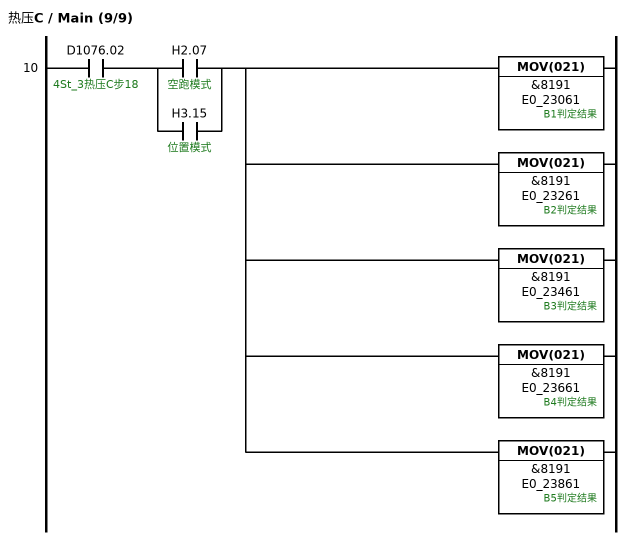
; [picture p216: 热压C / Main, rungs 10-10]
; rung 10
LD D1076.02  ; 4St_3热压C步18
LD H2.07  ; 空跑模式
OR H3.15  ; 位置模式
ANDLD
MOV(021) &8191 E0_23061  ; B1判定结果
MOV(021) &8191 E0_23261  ; B2判定结果
MOV(021) &8191 E0_23461  ; B3判定结果
MOV(021) &8191 E0_23661  ; B4判定结果
MOV(021) &8191 E0_23861  ; B5判定结果

### Section _4ST_3热压C

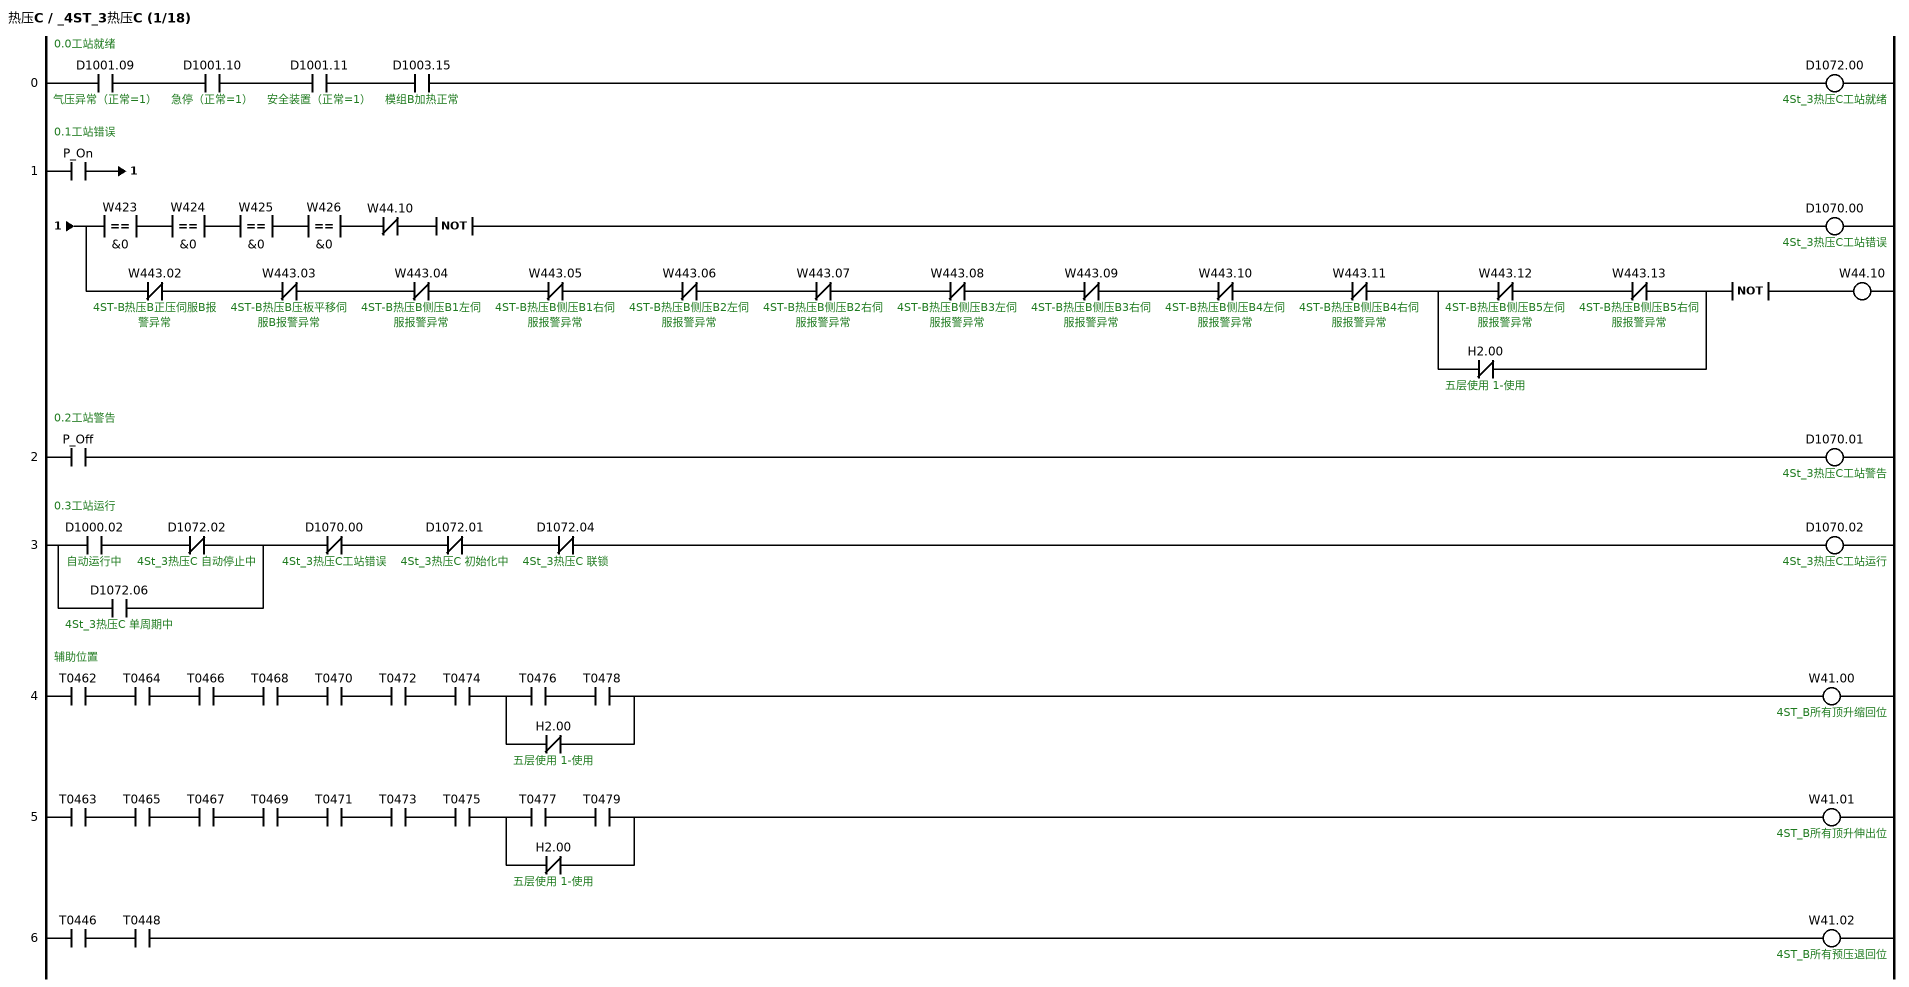
; rung 0: 0.0工站就绪
LD D1001.09  ; 气压异常（正常=1）
AND D1001.10  ; 急停（正常=1）
AND D1001.11  ; 安全装置（正常=1）
AND D1003.15  ; 模组B加热正常
OUT D1072.00  ; 4St_3热压C工站就绪
; rung 1: 0.1工站错误
LD P_On
OUT TR0
AND=(300) W423 &0
AND=(300) W424 &0
AND=(300) W425 &0
AND=(300) W426 &0
ANDNOT W44.10
NOT(520)
OUT D1070.00  ; 4St_3热压C工站错误
LD TR0
ANDNOT W443.02  ; 4ST-B热压B正压伺服B报警异常
ANDNOT W443.03  ; 4ST-B热压B压板平移伺服B报警异常
ANDNOT W443.04  ; 4ST-B热压B侧压B1左伺服报警异常
ANDNOT W443.05  ; 4ST-B热压B侧压B1右伺服报警异常
ANDNOT W443.06  ; 4ST-B热压B侧压B2左伺服报警异常
ANDNOT W443.07  ; 4ST-B热压B侧压B2右伺服报警异常
ANDNOT W443.08  ; 4ST-B热压B侧压B3左伺服报警异常
ANDNOT W443.09  ; 4ST-B热压B侧压B3右伺服报警异常
ANDNOT W443.10  ; 4ST-B热压B侧压B4左伺服报警异常
ANDNOT W443.11  ; 4ST-B热压B侧压B4右伺服报警异常
LDNOT W443.12  ; 4ST-B热压B侧压B5左伺服报警异常
ANDNOT W443.13  ; 4ST-B热压B侧压B5右伺服报警异常
ORNOT H2.00  ; 五层使用 1-使用
ANDLD
NOT(520)
OUT W44.10
; rung 2: 0.2工站警告
LD P_Off
OUT D1070.01  ; 4St_3热压C工站警告
; rung 3: 0.3工站运行
LD D1000.02  ; 自动运行中
ANDNOT D1072.02  ; 4St_3热压C 自动停止中
OR D1072.06  ; 4St_3热压C 单周期中
ANDNOT D1070.00  ; 4St_3热压C工站错误
ANDNOT D1072.01  ; 4St_3热压C 初始化中
ANDNOT D1072.04  ; 4St_3热压C 联锁
OUT D1070.02  ; 4St_3热压C工站运行
; rung 4: 辅助位置
LD T0462
AND T0464
AND T0466
AND T0468
AND T0470
AND T0472
AND T0474
LD T0476
AND T0478
ORNOT H2.00  ; 五层使用 1-使用
ANDLD
OUT W41.00  ; 4ST_B所有顶升缩回位
; rung 5
LD T0463
AND T0465
AND T0467
AND T0469
AND T0471
AND T0473
AND T0475
LD T0477
AND T0479
ORNOT H2.00  ; 五层使用 1-使用
ANDLD
OUT W41.01  ; 4ST_B所有顶升伸出位
; rung 6
LD T0446
AND T0448
OUT W41.02  ; 4ST_B所有预压退回位

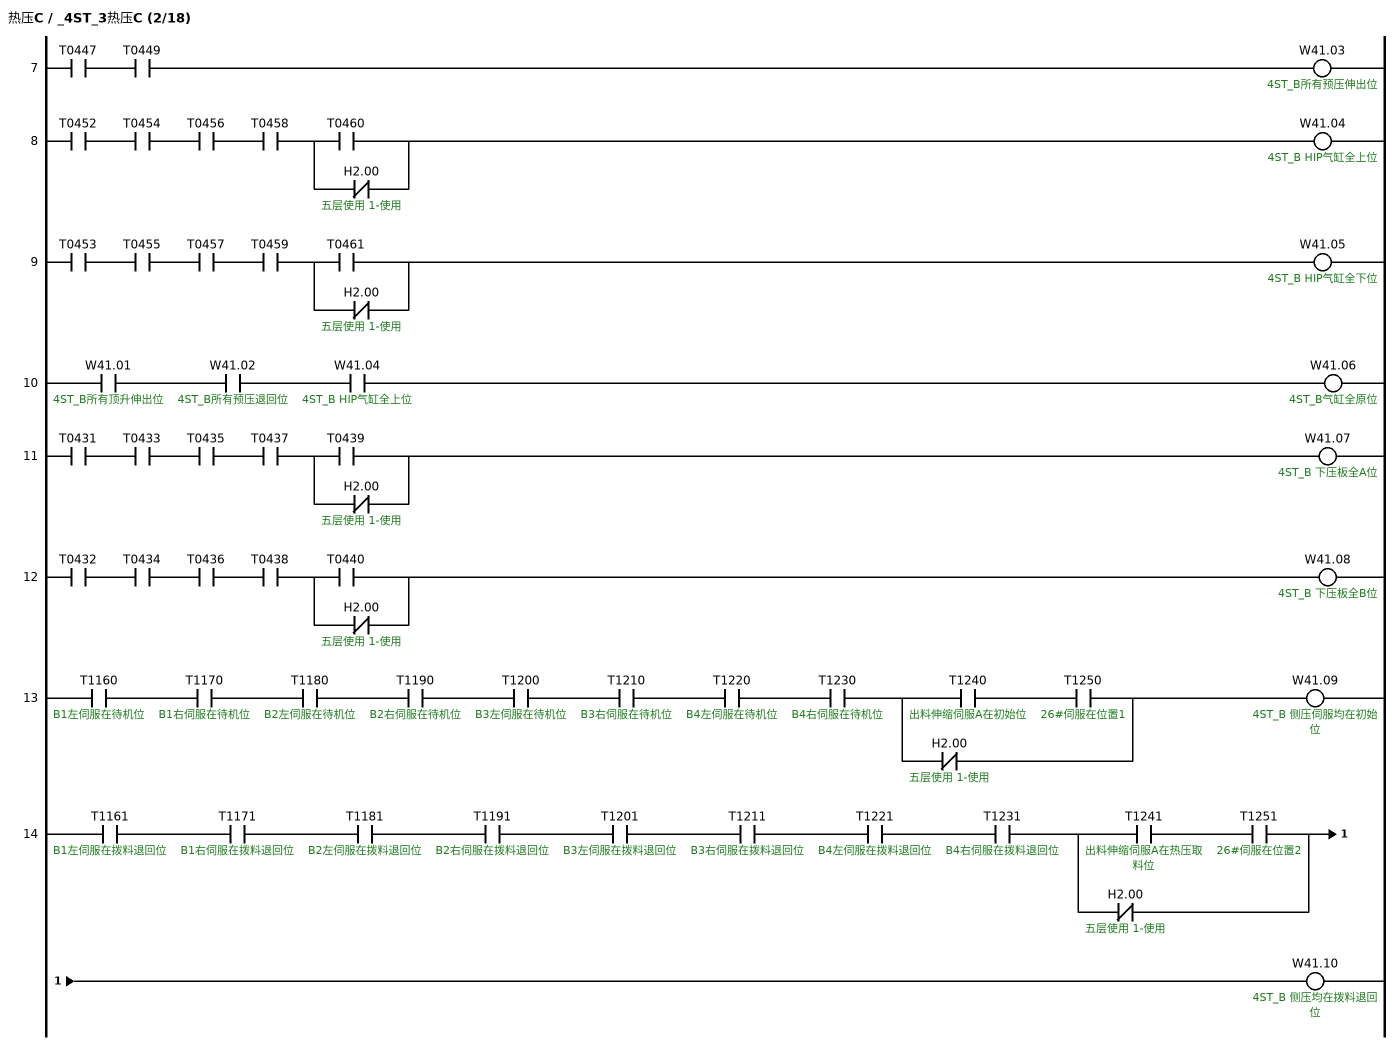
; rung 7
LD T0447
AND T0449
OUT W41.03  ; 4ST_B所有预压伸出位
; rung 8
LD T0452
AND T0454
AND T0456
AND T0458
LD T0460
ORNOT H2.00  ; 五层使用 1-使用
ANDLD
OUT W41.04  ; 4ST_B HIP气缸全上位
; rung 9
LD T0453
AND T0455
AND T0457
AND T0459
LD T0461
ORNOT H2.00  ; 五层使用 1-使用
ANDLD
OUT W41.05  ; 4ST_B HIP气缸全下位
; rung 10
LD W41.01  ; 4ST_B所有顶升伸出位
AND W41.02  ; 4ST_B所有预压退回位
AND W41.04  ; 4ST_B HIP气缸全上位
OUT W41.06  ; 4ST_B气缸全原位
; rung 11
LD T0431
AND T0433
AND T0435
AND T0437
LD T0439
ORNOT H2.00  ; 五层使用 1-使用
ANDLD
OUT W41.07  ; 4ST_B 下压板全A位
; rung 12
LD T0432
AND T0434
AND T0436
AND T0438
LD T0440
ORNOT H2.00  ; 五层使用 1-使用
ANDLD
OUT W41.08  ; 4ST_B 下压板全B位
; rung 13
LD T1160  ; B1左伺服在待机位
AND T1170  ; B1右伺服在待机位
AND T1180  ; B2左伺服在待机位
AND T1190  ; B2右伺服在待机位
AND T1200  ; B3左伺服在待机位
AND T1210  ; B3右伺服在待机位
AND T1220  ; B4左伺服在待机位
AND T1230  ; B4右伺服在待机位
LD T1240  ; 出料伸缩伺服A在初始位
AND T1250  ; 26#伺服在位置1
ORNOT H2.00  ; 五层使用 1-使用
ANDLD
OUT W41.09  ; 4ST_B 侧压伺服均在初始位
; rung 14
LD T1161  ; B1左伺服在拨料退回位
AND T1171  ; B1右伺服在拨料退回位
AND T1181  ; B2左伺服在拨料退回位
AND T1191  ; B2右伺服在拨料退回位
AND T1201  ; B3左伺服在拨料退回位
AND T1211  ; B3右伺服在拨料退回位
AND T1221  ; B4左伺服在拨料退回位
AND T1231  ; B4右伺服在拨料退回位
LD T1241  ; 出料伸缩伺服A在热压取料位
AND T1251  ; 26#伺服在位置2
ORNOT H2.00  ; 五层使用 1-使用
ANDLD
OUT W41.10  ; 4ST_B 侧压均在拨料退回位

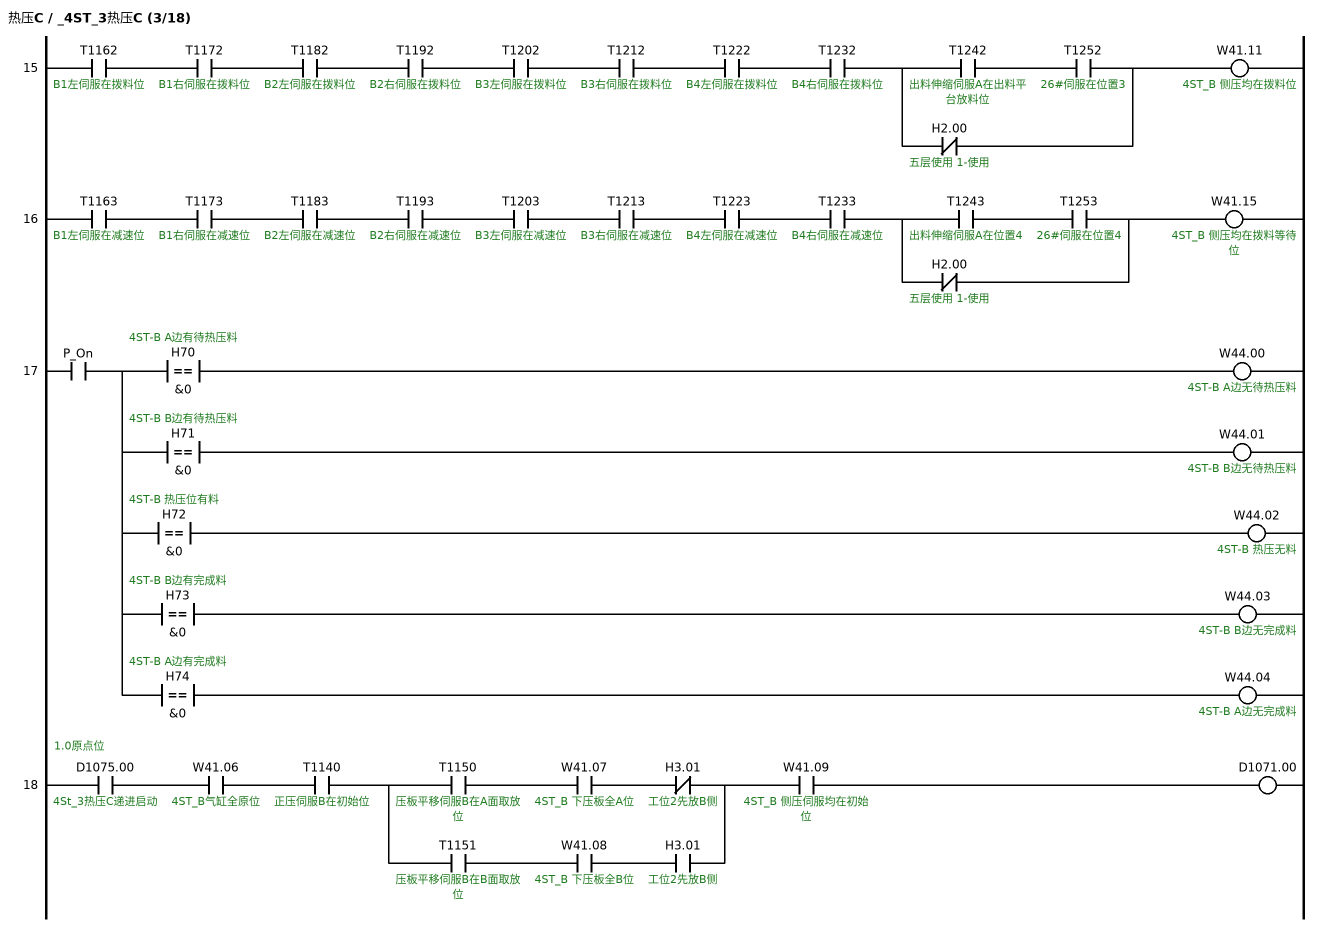
; rung 15
LD T1162  ; B1左伺服在拨料位
AND T1172  ; B1右伺服在拨料位
AND T1182  ; B2左伺服在拨料位
AND T1192  ; B2右伺服在拨料位
AND T1202  ; B3左伺服在拨料位
AND T1212  ; B3右伺服在拨料位
AND T1222  ; B4左伺服在拨料位
AND T1232  ; B4右伺服在拨料位
LD T1242  ; 出料伸缩伺服A在出料平台放料位
AND T1252  ; 26#伺服在位置3
ORNOT H2.00  ; 五层使用 1-使用
ANDLD
OUT W41.11  ; 4ST_B 侧压均在拨料位
; rung 16
LD T1163  ; B1左伺服在减速位
AND T1173  ; B1右伺服在减速位
AND T1183  ; B2左伺服在减速位
AND T1193  ; B2右伺服在减速位
AND T1203  ; B3左伺服在减速位
AND T1213  ; B3右伺服在减速位
AND T1223  ; B4左伺服在减速位
AND T1233  ; B4右伺服在减速位
LD T1243  ; 出料伸缩伺服A在位置4
AND T1253  ; 26#伺服在位置4
ORNOT H2.00  ; 五层使用 1-使用
ANDLD
OUT W41.15  ; 4ST_B 侧压均在拨料等待位
; rung 17
LD P_On
OUT TR0
AND=(300) H70 &0  ; 4ST-B A边有待热压料
OUT W44.00  ; 4ST-B A边无待热压料
LD TR0
AND=(300) H71 &0  ; 4ST-B B边有待热压料
OUT W44.01  ; 4ST-B B边无待热压料
LD TR0
AND=(300) H72 &0  ; 4ST-B 热压位有料
OUT W44.02  ; 4ST-B 热压无料
LD TR0
AND=(300) H73 &0  ; 4ST-B B边有完成料
OUT W44.03  ; 4ST-B B边无完成料
LD TR0
AND=(300) H74 &0  ; 4ST-B A边有完成料
OUT W44.04  ; 4ST-B A边无完成料
; rung 18: 1.0原点位
LD D1075.00  ; 4St_3热压C递进启动
AND W41.06  ; 4ST_B气缸全原位
AND T1140  ; 正压伺服B在初始位
LD T1150  ; 压板平移伺服B在A面取放位
AND W41.07  ; 4ST_B 下压板全A位
ANDNOT H3.01  ; 工位2先放B侧
LD T1151  ; 压板平移伺服B在B面取放位
AND W41.08  ; 4ST_B 下压板全B位
AND H3.01  ; 工位2先放B侧
ORLD
ANDLD
AND W41.09  ; 4ST_B 侧压伺服均在初始位
OUT D1071.00

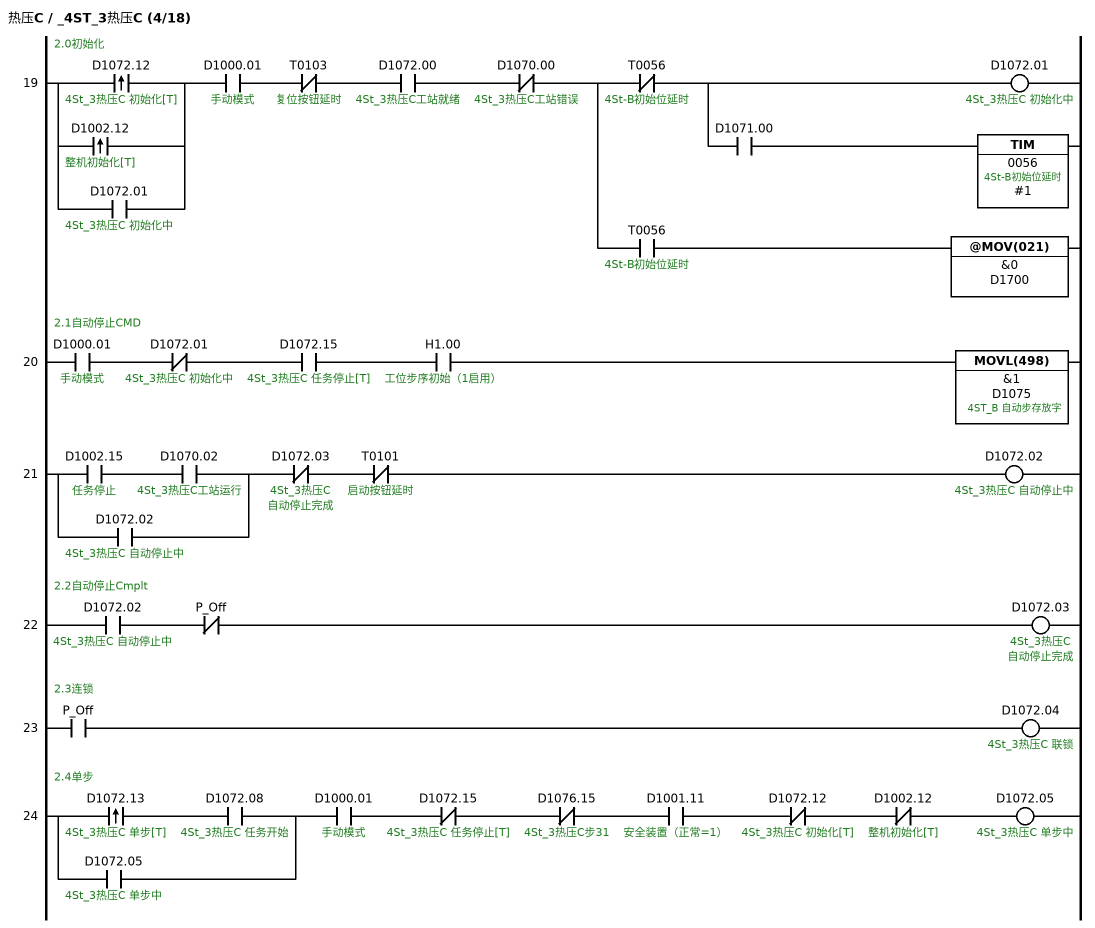
; rung 19: 2.0初始化
@LD D1072.12  ; 4St_3热压C 初始化[T]
@OR D1002.12  ; 整机初始化[T]
OR D1072.01  ; 4St_3热压C 初始化中
AND D1000.01  ; 手动模式
ANDNOT T0103  ; 复位按钮延时
AND D1072.00  ; 4St_3热压C工站就绪
ANDNOT D1070.00  ; 4St_3热压C工站错误
OUT TR0
ANDNOT T0056  ; 4St-B初始位延时
OUT D1072.01  ; 4St_3热压C 初始化中
AND D1071.00
TIM 0056 #1  ; 4St-B初始位延时
LD TR0
AND T0056  ; 4St-B初始位延时
@MOV(021) &0 D1700
; rung 20: 2.1自动停止CMD
LD D1000.01  ; 手动模式
ANDNOT D1072.01  ; 4St_3热压C 初始化中
AND D1072.15  ; 4St_3热压C 任务停止[T]
AND H1.00  ; 工位步序初始（1启用）
MOVL(498) &1 D1075  ; 4ST_B 自动步存放字
; rung 21
LD D1002.15  ; 任务停止
AND D1070.02  ; 4St_3热压C工站运行
OR D1072.02  ; 4St_3热压C 自动停止中
ANDNOT D1072.03  ; 4St_3热压C 自动停止完成
ANDNOT T0101  ; 启动按钮延时
OUT D1072.02  ; 4St_3热压C 自动停止中
; rung 22: 2.2自动停止Cmplt
LD D1072.02  ; 4St_3热压C 自动停止中
ANDNOT P_Off
OUT D1072.03  ; 4St_3热压C 自动停止完成
; rung 23: 2.3连锁
LD P_Off
OUT D1072.04  ; 4St_3热压C 联锁
; rung 24: 2.4单步
@LD D1072.13  ; 4St_3热压C 单步[T]
AND D1072.08  ; 4St_3热压C 任务开始
OR D1072.05  ; 4St_3热压C 单步中
AND D1000.01  ; 手动模式
ANDNOT D1072.15  ; 4St_3热压C 任务停止[T]
ANDNOT D1076.15  ; 4St_3热压C步31
AND D1001.11  ; 安全装置（正常=1）
ANDNOT D1072.12  ; 4St_3热压C 初始化[T]
ANDNOT D1002.12  ; 整机初始化[T]
OUT D1072.05  ; 4St_3热压C 单步中

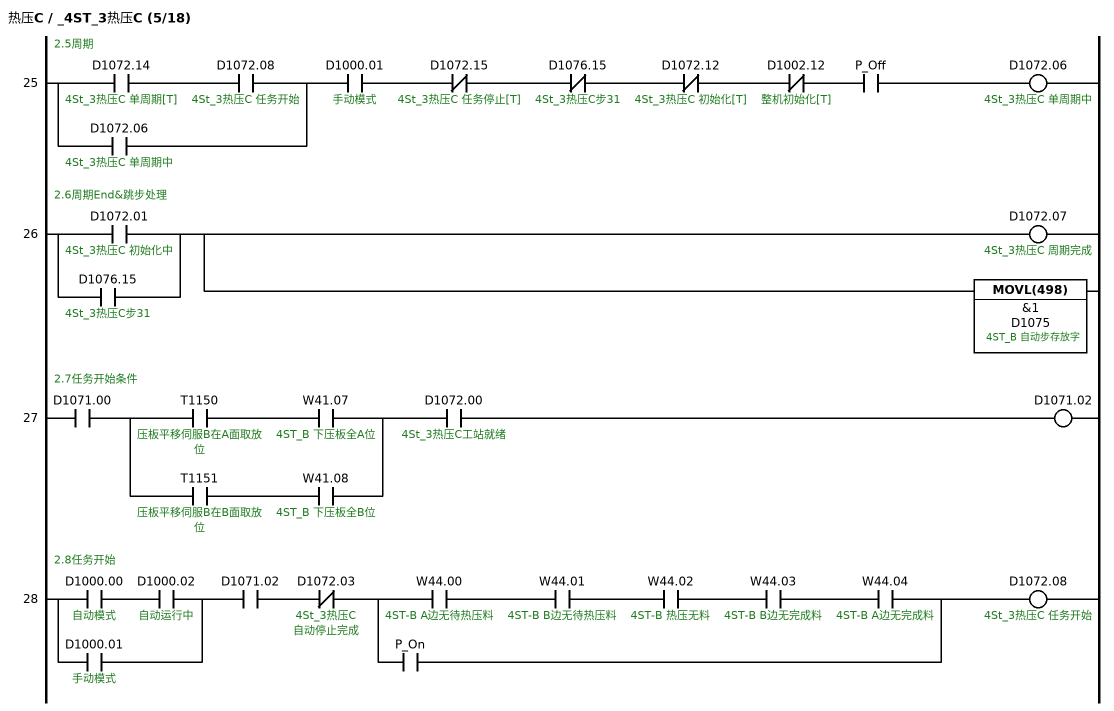
; rung 25: 2.5周期
LD D1072.14  ; 4St_3热压C 单周期[T]
AND D1072.08  ; 4St_3热压C 任务开始
OR D1072.06  ; 4St_3热压C 单周期中
AND D1000.01  ; 手动模式
ANDNOT D1072.15  ; 4St_3热压C 任务停止[T]
ANDNOT D1076.15  ; 4St_3热压C步31
ANDNOT D1072.12  ; 4St_3热压C 初始化[T]
ANDNOT D1002.12  ; 整机初始化[T]
AND P_Off
OUT D1072.06  ; 4St_3热压C 单周期中
; rung 26: 2.6周期End&跳步处理
LD D1072.01  ; 4St_3热压C 初始化中
OR D1076.15  ; 4St_3热压C步31
OUT D1072.07  ; 4St_3热压C 周期完成
MOVL(498) &1 D1075  ; 4ST_B 自动步存放字
; rung 27: 2.7任务开始条件
LD D1071.00
LD T1150  ; 压板平移伺服B在A面取放位
AND W41.07  ; 4ST_B 下压板全A位
LD T1151  ; 压板平移伺服B在B面取放位
AND W41.08  ; 4ST_B 下压板全B位
ORLD
ANDLD
AND D1072.00  ; 4St_3热压C工站就绪
OUT D1071.02
; rung 28: 2.8任务开始
LD D1000.00  ; 自动模式
AND D1000.02  ; 自动运行中
OR D1000.01  ; 手动模式
AND D1071.02
ANDNOT D1072.03  ; 4St_3热压C 自动停止完成
LD W44.00  ; 4ST-B A边无待热压料
AND W44.01  ; 4ST-B B边无待热压料
AND W44.02  ; 4ST-B 热压无料
AND W44.03  ; 4ST-B B边无完成料
AND W44.04  ; 4ST-B A边无完成料
OR P_On
ANDLD
OUT D1072.08  ; 4St_3热压C 任务开始

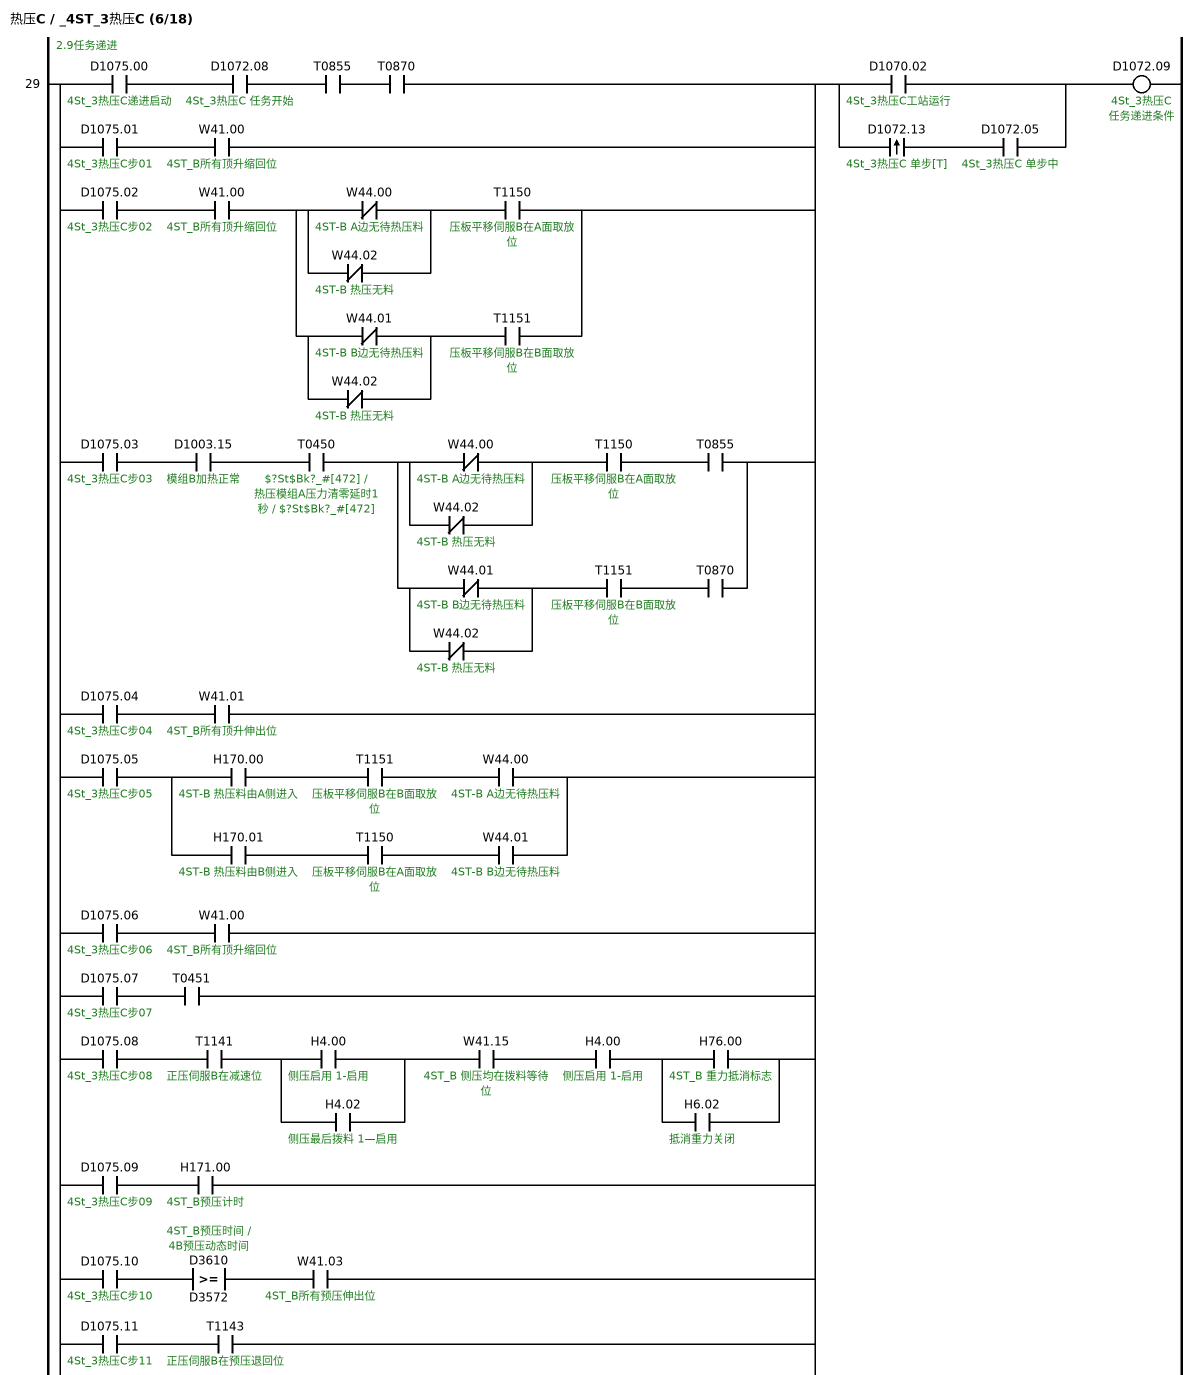

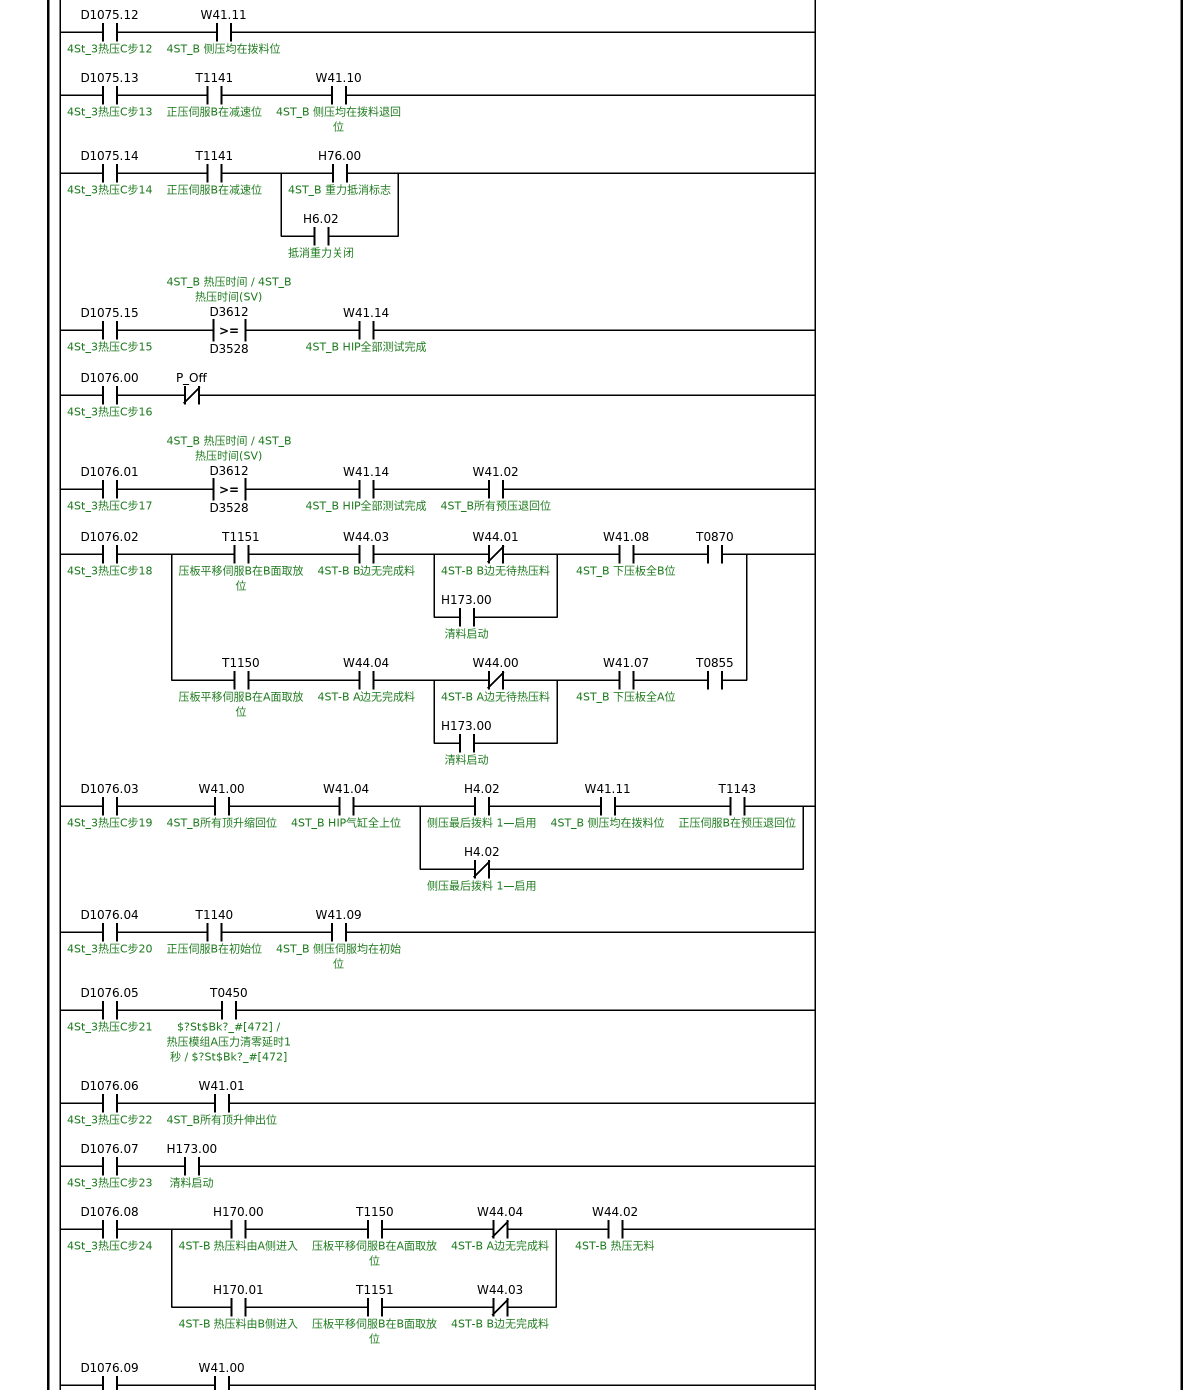

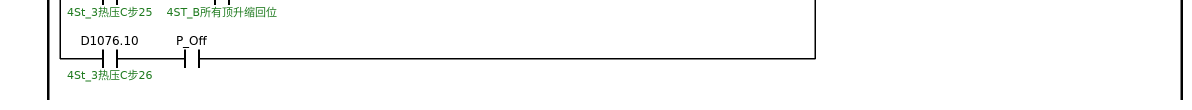
; rung 29: 2.9任务递进
LD D1075.00  ; 4St_3热压C递进启动
AND D1072.08  ; 4St_3热压C 任务开始
AND T0855
AND T0870
LD D1075.01  ; 4St_3热压C步01
AND W41.00  ; 4ST_B所有顶升缩回位
ORLD
LD D1075.02  ; 4St_3热压C步02
AND W41.00  ; 4ST_B所有顶升缩回位
LDNOT W44.00  ; 4ST-B A边无待热压料
ORNOT W44.02  ; 4ST-B 热压无料
AND T1150  ; 压板平移伺服B在A面取放位
LDNOT W44.01  ; 4ST-B B边无待热压料
ORNOT W44.02  ; 4ST-B 热压无料
AND T1151  ; 压板平移伺服B在B面取放位
ORLD
ANDLD
ORLD
LD D1075.03  ; 4St_3热压C步03
AND D1003.15  ; 模组B加热正常
AND T0450  ; $?St$Bk?_#[472] / 热压模组A压力清零延时1秒 / $?St$Bk?_#[472]
LDNOT W44.00  ; 4ST-B A边无待热压料
ORNOT W44.02  ; 4ST-B 热压无料
AND T1150  ; 压板平移伺服B在A面取放位
AND T0855
LDNOT W44.01  ; 4ST-B B边无待热压料
ORNOT W44.02  ; 4ST-B 热压无料
AND T1151  ; 压板平移伺服B在B面取放位
AND T0870
ORLD
ANDLD
ORLD
LD D1075.04  ; 4St_3热压C步04
AND W41.01  ; 4ST_B所有顶升伸出位
ORLD
LD D1075.05  ; 4St_3热压C步05
LD H170.00  ; 4ST-B 热压料由A侧进入
AND T1151  ; 压板平移伺服B在B面取放位
AND W44.00  ; 4ST-B A边无待热压料
LD H170.01  ; 4ST-B 热压料由B侧进入
AND T1150  ; 压板平移伺服B在A面取放位
AND W44.01  ; 4ST-B B边无待热压料
ORLD
ANDLD
ORLD
LD D1075.06  ; 4St_3热压C步06
AND W41.00  ; 4ST_B所有顶升缩回位
ORLD
LD D1075.07  ; 4St_3热压C步07
AND T0451
ORLD
LD D1075.08  ; 4St_3热压C步08
AND T1141  ; 正压伺服B在减速位
LD H4.00  ; 侧压启用 1-启用
OR H4.02  ; 侧压最后拨料 1—启用
ANDLD
AND W41.15  ; 4ST_B 侧压均在拨料等待位
AND H4.00  ; 侧压启用 1-启用
LD H76.00  ; 4ST_B 重力抵消标志
OR H6.02  ; 抵消重力关闭
ANDLD
ORLD
LD D1075.09  ; 4St_3热压C步09
AND H171.00  ; 4ST_B预压计时
ORLD
LD D1075.10  ; 4St_3热压C步10
AND>=(325) D3610 D3572  ; 4ST_B预压时间, 4B预压动态时间
AND W41.03  ; 4ST_B所有预压伸出位
ORLD
LD D1075.11  ; 4St_3热压C步11
AND T1143  ; 正压伺服B在预压退回位
ORLD
LD D1075.12  ; 4St_3热压C步12
AND W41.11  ; 4ST_B 侧压均在拨料位
ORLD
LD D1075.13  ; 4St_3热压C步13
AND T1141  ; 正压伺服B在减速位
AND W41.10  ; 4ST_B 侧压均在拨料退回位
ORLD
LD D1075.14  ; 4St_3热压C步14
AND T1141  ; 正压伺服B在减速位
LD H76.00  ; 4ST_B 重力抵消标志
OR H6.02  ; 抵消重力关闭
ANDLD
ORLD
LD D1075.15  ; 4St_3热压C步15
AND>=(325) D3612 D3528  ; 4ST_B 热压时间, 4ST_B 热压时间(SV)
AND W41.14  ; 4ST_B HIP全部测试完成
ORLD
LD D1076.00  ; 4St_3热压C步16
ANDNOT P_Off
ORLD
LD D1076.01  ; 4St_3热压C步17
AND>=(325) D3612 D3528  ; 4ST_B 热压时间, 4ST_B 热压时间(SV)
AND W41.14  ; 4ST_B HIP全部测试完成
AND W41.02  ; 4ST_B所有预压退回位
ORLD
LD D1076.02  ; 4St_3热压C步18
LD T1151  ; 压板平移伺服B在B面取放位
AND W44.03  ; 4ST-B B边无完成料
LDNOT W44.01  ; 4ST-B B边无待热压料
OR H173.00  ; 清料启动
ANDLD
AND W41.08  ; 4ST_B 下压板全B位
AND T0870
LD T1150  ; 压板平移伺服B在A面取放位
AND W44.04  ; 4ST-B A边无完成料
LDNOT W44.00  ; 4ST-B A边无待热压料
OR H173.00  ; 清料启动
ANDLD
AND W41.07  ; 4ST_B 下压板全A位
AND T0855
ORLD
ANDLD
ORLD
LD D1076.03  ; 4St_3热压C步19
AND W41.00  ; 4ST_B所有顶升缩回位
AND W41.04  ; 4ST_B HIP气缸全上位
LD H4.02  ; 侧压最后拨料 1—启用
AND W41.11  ; 4ST_B 侧压均在拨料位
AND T1143  ; 正压伺服B在预压退回位
ORNOT H4.02  ; 侧压最后拨料 1—启用
ANDLD
ORLD
LD D1076.04  ; 4St_3热压C步20
AND T1140  ; 正压伺服B在初始位
AND W41.09  ; 4ST_B 侧压伺服均在初始位
ORLD
LD D1076.05  ; 4St_3热压C步21
AND T0450  ; $?St$Bk?_#[472] / 热压模组A压力清零延时1秒 / $?St$Bk?_#[472]
ORLD
LD D1076.06  ; 4St_3热压C步22
AND W41.01  ; 4ST_B所有顶升伸出位
ORLD
LD D1076.07  ; 4St_3热压C步23
AND H173.00  ; 清料启动
ORLD
LD D1076.08  ; 4St_3热压C步24
LD H170.00  ; 4ST-B 热压料由A侧进入
AND T1150  ; 压板平移伺服B在A面取放位
ANDNOT W44.04  ; 4ST-B A边无完成料
LD H170.01  ; 4ST-B 热压料由B侧进入
AND T1151  ; 压板平移伺服B在B面取放位
ANDNOT W44.03  ; 4ST-B B边无完成料
ORLD
ANDLD
AND W44.02  ; 4ST-B 热压无料
ORLD
LD D1076.09  ; 4St_3热压C步25
AND W41.00  ; 4ST_B所有顶升缩回位
ORLD
LD D1076.10  ; 4St_3热压C步26
AND P_Off
ORLD
LD D1070.02  ; 4St_3热压C工站运行
@LD D1072.13  ; 4St_3热压C 单步[T]
AND D1072.05  ; 4St_3热压C 单步中
ORLD
ANDLD
OUT D1072.09  ; 4St_3热压C 任务递进条件

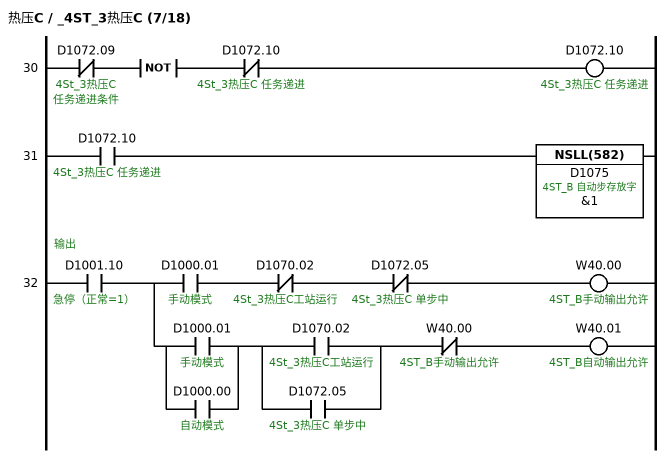
; rung 30
LDNOT D1072.09  ; 4St_3热压C 任务递进条件
NOT(520)
ANDNOT D1072.10  ; 4St_3热压C 任务递进
OUT D1072.10  ; 4St_3热压C 任务递进
; rung 31
LD D1072.10  ; 4St_3热压C 任务递进
NSLL(582) D1075 &1  ; 4ST_B 自动步存放字
; rung 32: 输出
LD D1001.10  ; 急停（正常=1）
OUT TR0
AND D1000.01  ; 手动模式
ANDNOT D1070.02  ; 4St_3热压C工站运行
ANDNOT D1072.05  ; 4St_3热压C 单步中
OUT W40.00  ; 4ST_B手动输出允许
LD TR0
LD D1000.01  ; 手动模式
OR D1000.00  ; 自动模式
ANDLD
LD D1070.02  ; 4St_3热压C工站运行
OR D1072.05  ; 4St_3热压C 单步中
ANDLD
ANDNOT W40.00  ; 4ST_B手动输出允许
OUT W40.01  ; 4ST_B自动输出允许

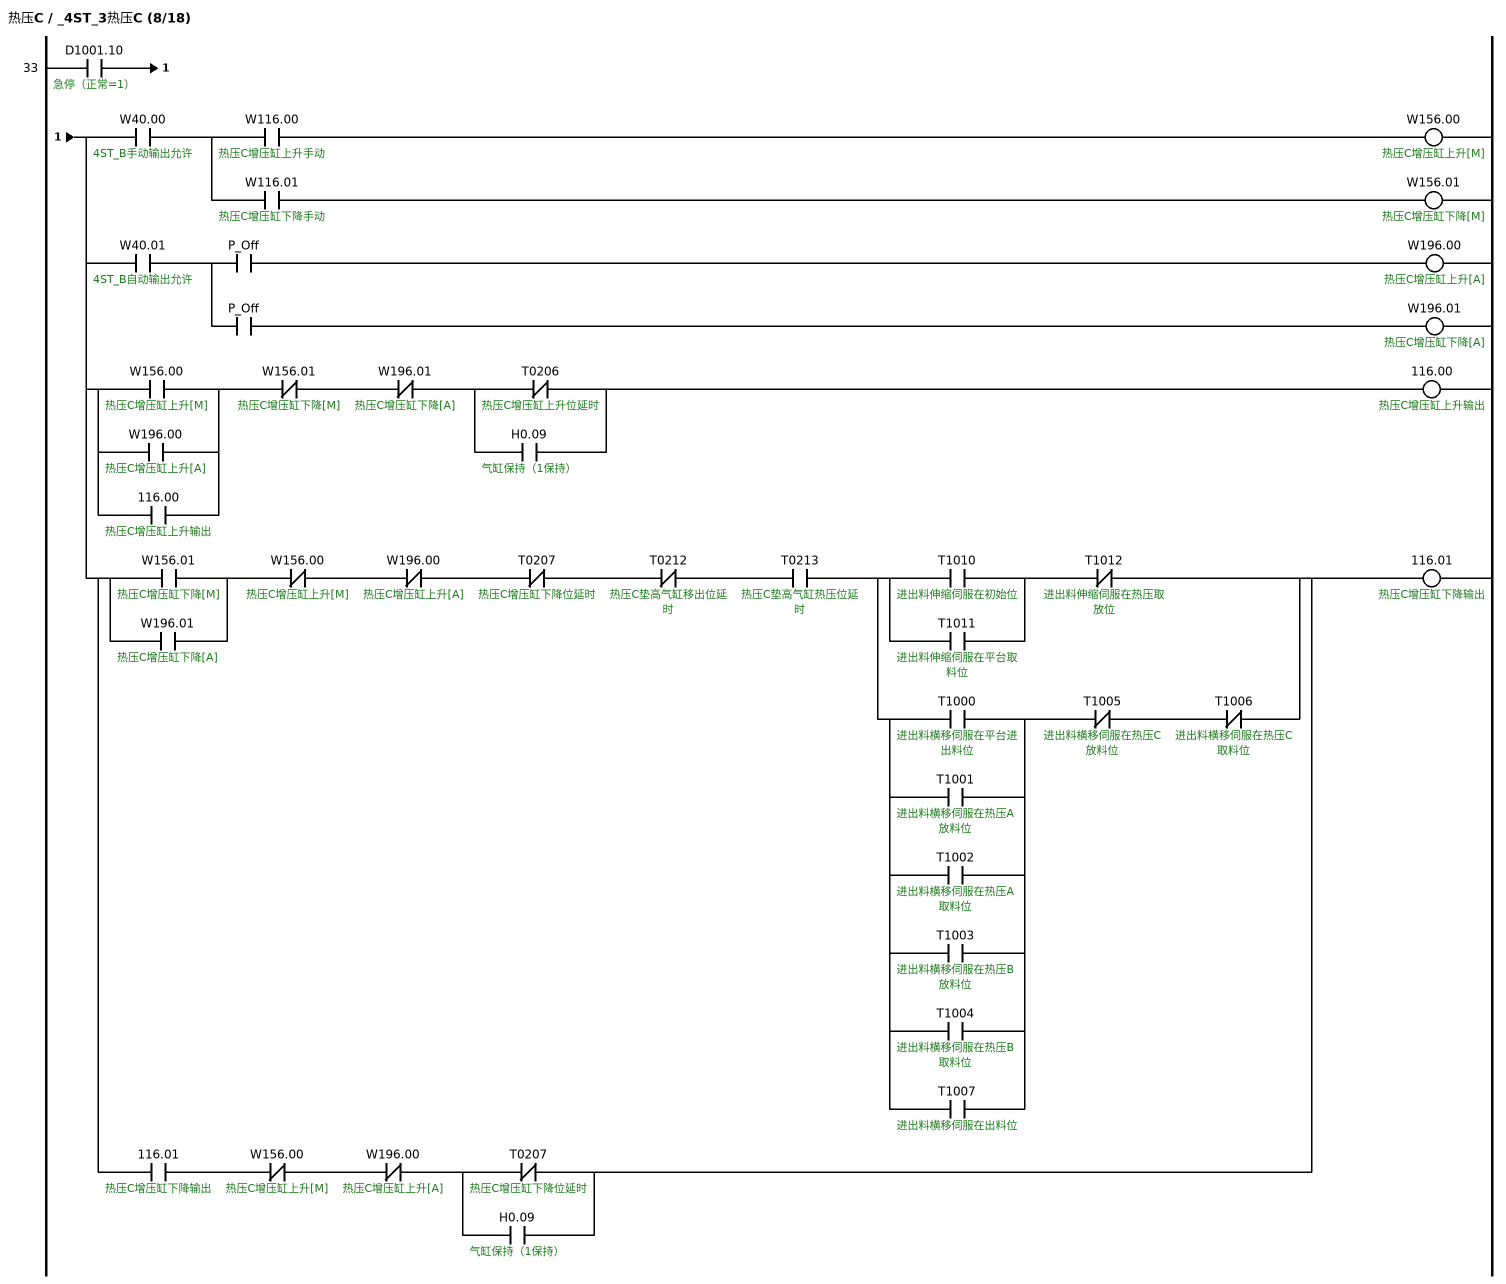
; rung 33
LD D1001.10  ; 急停（正常=1）
OUT TR0
AND W40.00  ; 4ST_B手动输出允许
OUT TR1
AND W116.00  ; 热压C增压缸上升手动
OUT W156.00  ; 热压C增压缸上升[M]
LD TR1
AND W116.01  ; 热压C增压缸下降手动
OUT W156.01  ; 热压C增压缸下降[M]
LD TR0
AND W40.01  ; 4ST_B自动输出允许
OUT TR1
AND P_Off
OUT W196.00  ; 热压C增压缸上升[A]
LD TR1
AND P_Off
OUT W196.01  ; 热压C增压缸下降[A]
LD TR0
LD W156.00  ; 热压C增压缸上升[M]
OR W196.00  ; 热压C增压缸上升[A]
OR 116.00  ; 热压C增压缸上升输出
ANDLD
ANDNOT W156.01  ; 热压C增压缸下降[M]
ANDNOT W196.01  ; 热压C增压缸下降[A]
LDNOT T0206  ; 热压C增压缸上升位延时
OR H0.09  ; 气缸保持（1保持）
ANDLD
OUT 116.00  ; 热压C增压缸上升输出
LD TR0
LD W156.01  ; 热压C增压缸下降[M]
OR W196.01  ; 热压C增压缸下降[A]
ANDNOT W156.00  ; 热压C增压缸上升[M]
ANDNOT W196.00  ; 热压C增压缸上升[A]
ANDNOT T0207  ; 热压C增压缸下降位延时
ANDNOT T0212  ; 热压C垫高气缸移出位延时
AND T0213  ; 热压C垫高气缸热压位延时
LD T1010  ; 进出料伸缩伺服在初始位
OR T1011  ; 进出料伸缩伺服在平台取料位
ANDNOT T1012  ; 进出料伸缩伺服在热压取放位
LD T1000  ; 进出料横移伺服在平台进出料位
OR T1001  ; 进出料横移伺服在热压A放料位
OR T1002  ; 进出料横移伺服在热压A取料位
OR T1003  ; 进出料横移伺服在热压B放料位
OR T1004  ; 进出料横移伺服在热压B取料位
OR T1007  ; 进出料横移伺服在出料位
ANDNOT T1005  ; 进出料横移伺服在热压C放料位
ANDNOT T1006  ; 进出料横移伺服在热压C取料位
ORLD
ANDLD
LD 116.01  ; 热压C增压缸下降输出
ANDNOT W156.00  ; 热压C增压缸上升[M]
ANDNOT W196.00  ; 热压C增压缸上升[A]
LDNOT T0207  ; 热压C增压缸下降位延时
OR H0.09  ; 气缸保持（1保持）
ANDLD
ORLD
ANDLD
OUT 116.01  ; 热压C增压缸下降输出

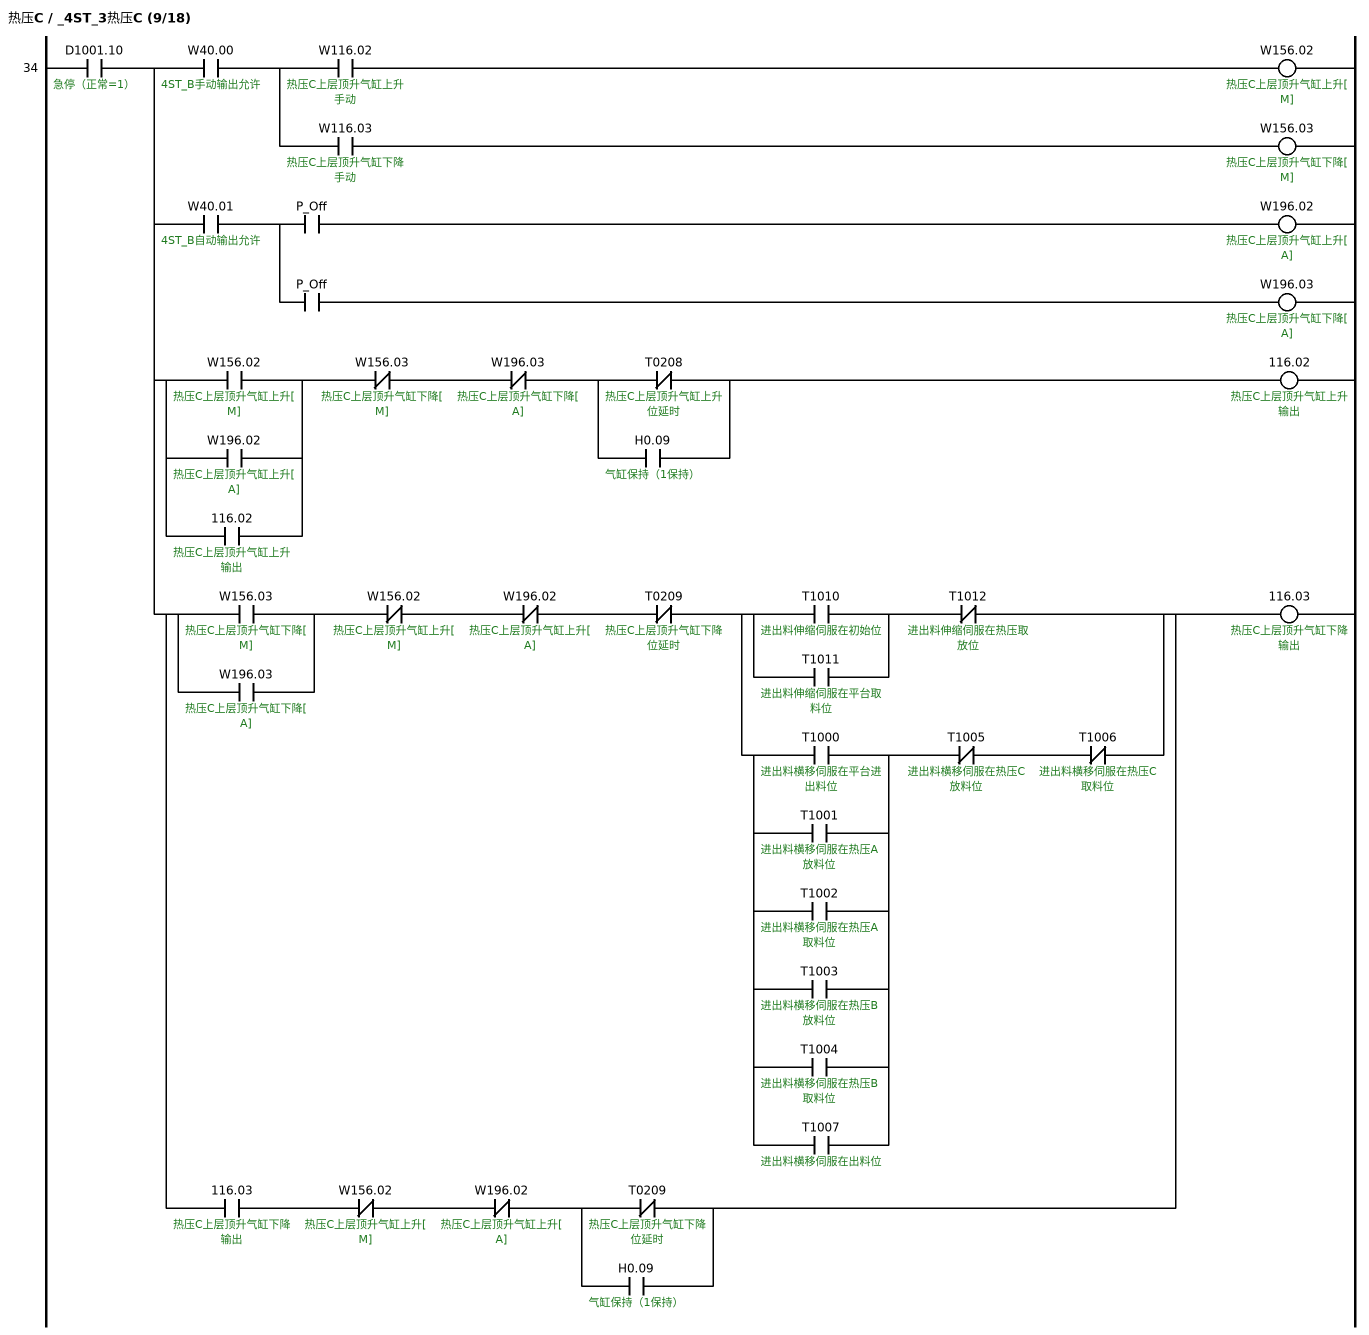
; rung 34
LD D1001.10  ; 急停（正常=1）
OUT TR0
AND W40.00  ; 4ST_B手动输出允许
OUT TR1
AND W116.02  ; 热压C上层顶升气缸上升手动
OUT W156.02  ; 热压C上层顶升气缸上升[M]
LD TR1
AND W116.03  ; 热压C上层顶升气缸下降手动
OUT W156.03  ; 热压C上层顶升气缸下降[M]
LD TR0
AND W40.01  ; 4ST_B自动输出允许
OUT TR1
AND P_Off
OUT W196.02  ; 热压C上层顶升气缸上升[A]
LD TR1
AND P_Off
OUT W196.03  ; 热压C上层顶升气缸下降[A]
LD TR0
LD W156.02  ; 热压C上层顶升气缸上升[M]
OR W196.02  ; 热压C上层顶升气缸上升[A]
OR 116.02  ; 热压C上层顶升气缸上升输出
ANDLD
ANDNOT W156.03  ; 热压C上层顶升气缸下降[M]
ANDNOT W196.03  ; 热压C上层顶升气缸下降[A]
LDNOT T0208  ; 热压C上层顶升气缸上升位延时
OR H0.09  ; 气缸保持（1保持）
ANDLD
OUT 116.02  ; 热压C上层顶升气缸上升输出
LD TR0
LD W156.03  ; 热压C上层顶升气缸下降[M]
OR W196.03  ; 热压C上层顶升气缸下降[A]
ANDNOT W156.02  ; 热压C上层顶升气缸上升[M]
ANDNOT W196.02  ; 热压C上层顶升气缸上升[A]
ANDNOT T0209  ; 热压C上层顶升气缸下降位延时
LD T1010  ; 进出料伸缩伺服在初始位
OR T1011  ; 进出料伸缩伺服在平台取料位
ANDNOT T1012  ; 进出料伸缩伺服在热压取放位
LD T1000  ; 进出料横移伺服在平台进出料位
OR T1001  ; 进出料横移伺服在热压A放料位
OR T1002  ; 进出料横移伺服在热压A取料位
OR T1003  ; 进出料横移伺服在热压B放料位
OR T1004  ; 进出料横移伺服在热压B取料位
OR T1007  ; 进出料横移伺服在出料位
ANDNOT T1005  ; 进出料横移伺服在热压C放料位
ANDNOT T1006  ; 进出料横移伺服在热压C取料位
ORLD
ANDLD
LD 116.03  ; 热压C上层顶升气缸下降输出
ANDNOT W156.02  ; 热压C上层顶升气缸上升[M]
ANDNOT W196.02  ; 热压C上层顶升气缸上升[A]
LDNOT T0209  ; 热压C上层顶升气缸下降位延时
OR H0.09  ; 气缸保持（1保持）
ANDLD
ORLD
ANDLD
OUT 116.03  ; 热压C上层顶升气缸下降输出

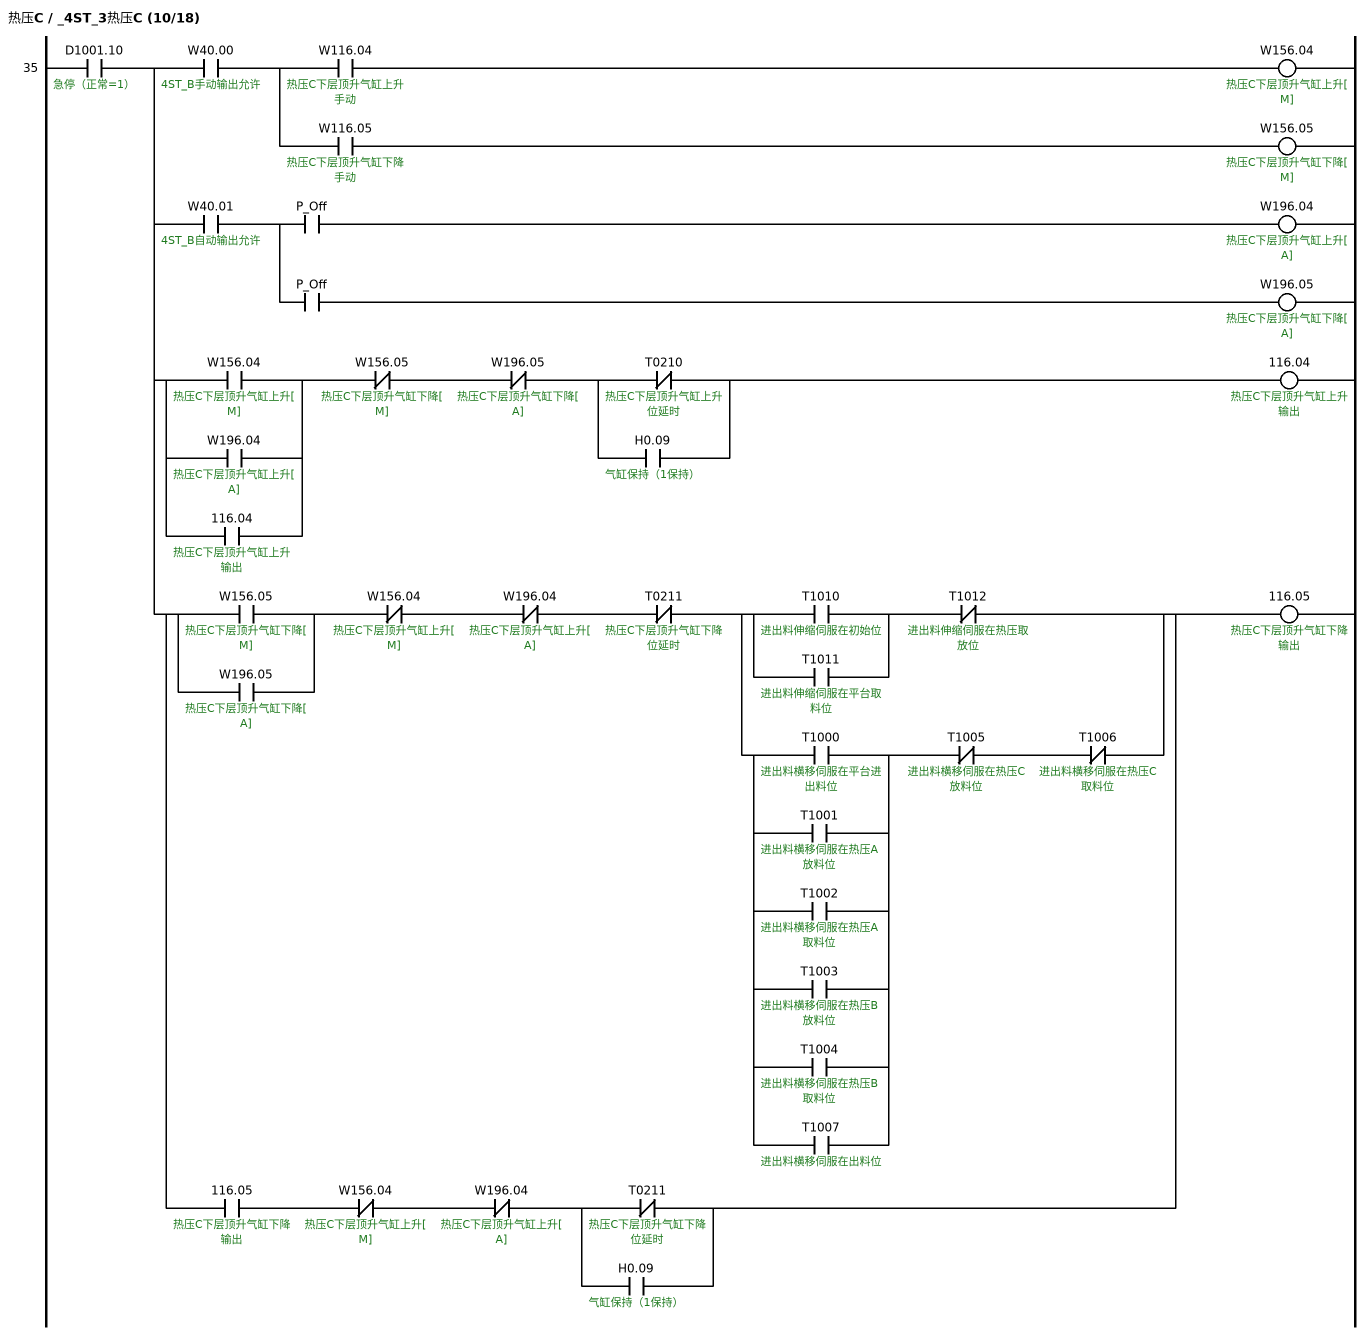
; rung 35
LD D1001.10  ; 急停（正常=1）
OUT TR0
AND W40.00  ; 4ST_B手动输出允许
OUT TR1
AND W116.04  ; 热压C下层顶升气缸上升手动
OUT W156.04  ; 热压C下层顶升气缸上升[M]
LD TR1
AND W116.05  ; 热压C下层顶升气缸下降手动
OUT W156.05  ; 热压C下层顶升气缸下降[M]
LD TR0
AND W40.01  ; 4ST_B自动输出允许
OUT TR1
AND P_Off
OUT W196.04  ; 热压C下层顶升气缸上升[A]
LD TR1
AND P_Off
OUT W196.05  ; 热压C下层顶升气缸下降[A]
LD TR0
LD W156.04  ; 热压C下层顶升气缸上升[M]
OR W196.04  ; 热压C下层顶升气缸上升[A]
OR 116.04  ; 热压C下层顶升气缸上升输出
ANDLD
ANDNOT W156.05  ; 热压C下层顶升气缸下降[M]
ANDNOT W196.05  ; 热压C下层顶升气缸下降[A]
LDNOT T0210  ; 热压C下层顶升气缸上升位延时
OR H0.09  ; 气缸保持（1保持）
ANDLD
OUT 116.04  ; 热压C下层顶升气缸上升输出
LD TR0
LD W156.05  ; 热压C下层顶升气缸下降[M]
OR W196.05  ; 热压C下层顶升气缸下降[A]
ANDNOT W156.04  ; 热压C下层顶升气缸上升[M]
ANDNOT W196.04  ; 热压C下层顶升气缸上升[A]
ANDNOT T0211  ; 热压C下层顶升气缸下降位延时
LD T1010  ; 进出料伸缩伺服在初始位
OR T1011  ; 进出料伸缩伺服在平台取料位
ANDNOT T1012  ; 进出料伸缩伺服在热压取放位
LD T1000  ; 进出料横移伺服在平台进出料位
OR T1001  ; 进出料横移伺服在热压A放料位
OR T1002  ; 进出料横移伺服在热压A取料位
OR T1003  ; 进出料横移伺服在热压B放料位
OR T1004  ; 进出料横移伺服在热压B取料位
OR T1007  ; 进出料横移伺服在出料位
ANDNOT T1005  ; 进出料横移伺服在热压C放料位
ANDNOT T1006  ; 进出料横移伺服在热压C取料位
ORLD
ANDLD
LD 116.05  ; 热压C下层顶升气缸下降输出
ANDNOT W156.04  ; 热压C下层顶升气缸上升[M]
ANDNOT W196.04  ; 热压C下层顶升气缸上升[A]
LDNOT T0211  ; 热压C下层顶升气缸下降位延时
OR H0.09  ; 气缸保持（1保持）
ANDLD
ORLD
ANDLD
OUT 116.05  ; 热压C下层顶升气缸下降输出

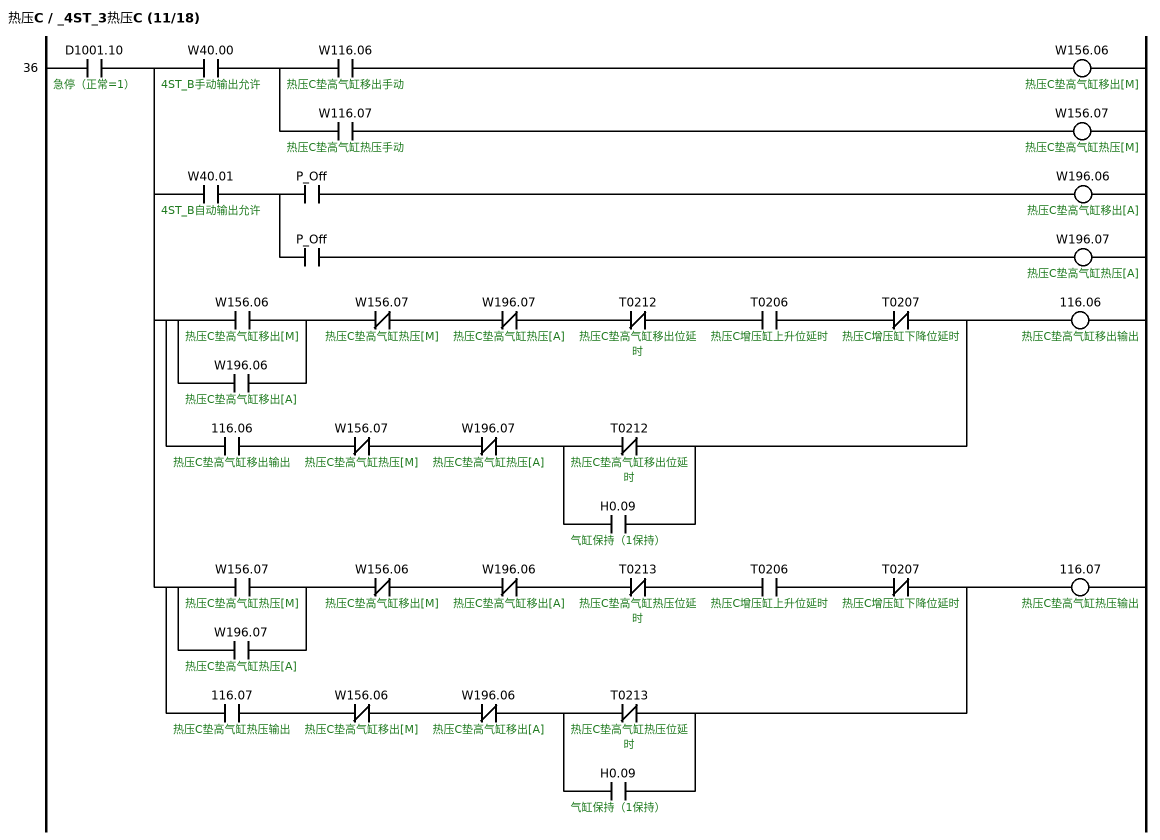
; rung 36
LD D1001.10  ; 急停（正常=1）
OUT TR0
AND W40.00  ; 4ST_B手动输出允许
OUT TR1
AND W116.06  ; 热压C垫高气缸移出手动
OUT W156.06  ; 热压C垫高气缸移出[M]
LD TR1
AND W116.07  ; 热压C垫高气缸热压手动
OUT W156.07  ; 热压C垫高气缸热压[M]
LD TR0
AND W40.01  ; 4ST_B自动输出允许
OUT TR1
AND P_Off
OUT W196.06  ; 热压C垫高气缸移出[A]
LD TR1
AND P_Off
OUT W196.07  ; 热压C垫高气缸热压[A]
LD TR0
LD W156.06  ; 热压C垫高气缸移出[M]
OR W196.06  ; 热压C垫高气缸移出[A]
ANDNOT W156.07  ; 热压C垫高气缸热压[M]
ANDNOT W196.07  ; 热压C垫高气缸热压[A]
ANDNOT T0212  ; 热压C垫高气缸移出位延时
AND T0206  ; 热压C增压缸上升位延时
ANDNOT T0207  ; 热压C增压缸下降位延时
LD 116.06  ; 热压C垫高气缸移出输出
ANDNOT W156.07  ; 热压C垫高气缸热压[M]
ANDNOT W196.07  ; 热压C垫高气缸热压[A]
LDNOT T0212  ; 热压C垫高气缸移出位延时
OR H0.09  ; 气缸保持（1保持）
ANDLD
ORLD
ANDLD
OUT 116.06  ; 热压C垫高气缸移出输出
LD TR0
LD W156.07  ; 热压C垫高气缸热压[M]
OR W196.07  ; 热压C垫高气缸热压[A]
ANDNOT W156.06  ; 热压C垫高气缸移出[M]
ANDNOT W196.06  ; 热压C垫高气缸移出[A]
ANDNOT T0213  ; 热压C垫高气缸热压位延时
AND T0206  ; 热压C增压缸上升位延时
ANDNOT T0207  ; 热压C增压缸下降位延时
LD 116.07  ; 热压C垫高气缸热压输出
ANDNOT W156.06  ; 热压C垫高气缸移出[M]
ANDNOT W196.06  ; 热压C垫高气缸移出[A]
LDNOT T0213  ; 热压C垫高气缸热压位延时
OR H0.09  ; 气缸保持（1保持）
ANDLD
ORLD
ANDLD
OUT 116.07  ; 热压C垫高气缸热压输出

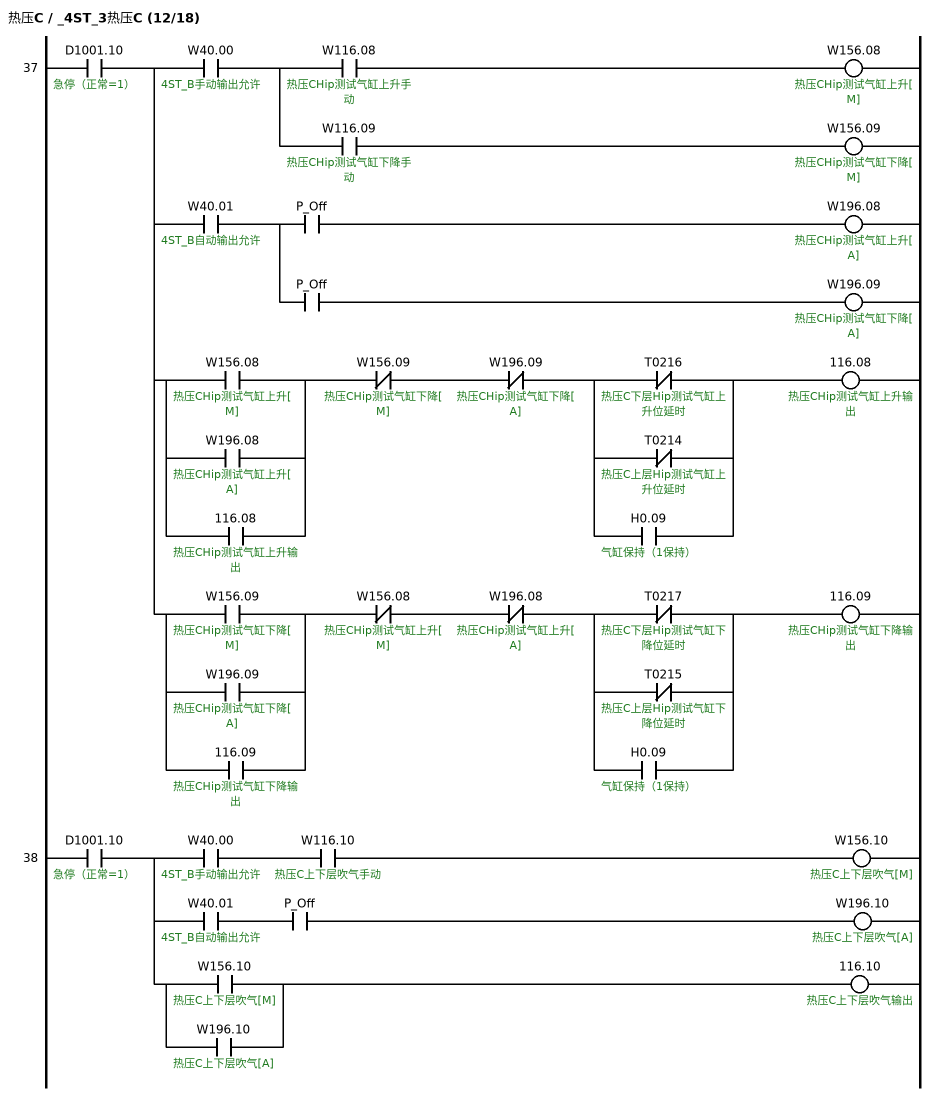
; rung 37
LD D1001.10  ; 急停（正常=1）
OUT TR0
AND W40.00  ; 4ST_B手动输出允许
OUT TR1
AND W116.08  ; 热压CHip测试气缸上升手动
OUT W156.08  ; 热压CHip测试气缸上升[M]
LD TR1
AND W116.09  ; 热压CHip测试气缸下降手动
OUT W156.09  ; 热压CHip测试气缸下降[M]
LD TR0
AND W40.01  ; 4ST_B自动输出允许
OUT TR1
AND P_Off
OUT W196.08  ; 热压CHip测试气缸上升[A]
LD TR1
AND P_Off
OUT W196.09  ; 热压CHip测试气缸下降[A]
LD TR0
LD W156.08  ; 热压CHip测试气缸上升[M]
OR W196.08  ; 热压CHip测试气缸上升[A]
OR 116.08  ; 热压CHip测试气缸上升输出
ANDLD
ANDNOT W156.09  ; 热压CHip测试气缸下降[M]
ANDNOT W196.09  ; 热压CHip测试气缸下降[A]
LDNOT T0216  ; 热压C下层Hip测试气缸上升位延时
ORNOT T0214  ; 热压C上层Hip测试气缸上升位延时
OR H0.09  ; 气缸保持（1保持）
ANDLD
OUT 116.08  ; 热压CHip测试气缸上升输出
LD TR0
LD W156.09  ; 热压CHip测试气缸下降[M]
OR W196.09  ; 热压CHip测试气缸下降[A]
OR 116.09  ; 热压CHip测试气缸下降输出
ANDLD
ANDNOT W156.08  ; 热压CHip测试气缸上升[M]
ANDNOT W196.08  ; 热压CHip测试气缸上升[A]
LDNOT T0217  ; 热压C下层Hip测试气缸下降位延时
ORNOT T0215  ; 热压C上层Hip测试气缸下降位延时
OR H0.09  ; 气缸保持（1保持）
ANDLD
OUT 116.09  ; 热压CHip测试气缸下降输出
; rung 38
LD D1001.10  ; 急停（正常=1）
OUT TR0
AND W40.00  ; 4ST_B手动输出允许
AND W116.10  ; 热压C上下层吹气手动
OUT W156.10  ; 热压C上下层吹气[M]
LD TR0
AND W40.01  ; 4ST_B自动输出允许
AND P_Off
OUT W196.10  ; 热压C上下层吹气[A]
LD TR0
LD W156.10  ; 热压C上下层吹气[M]
OR W196.10  ; 热压C上下层吹气[A]
ANDLD
OUT 116.10  ; 热压C上下层吹气输出

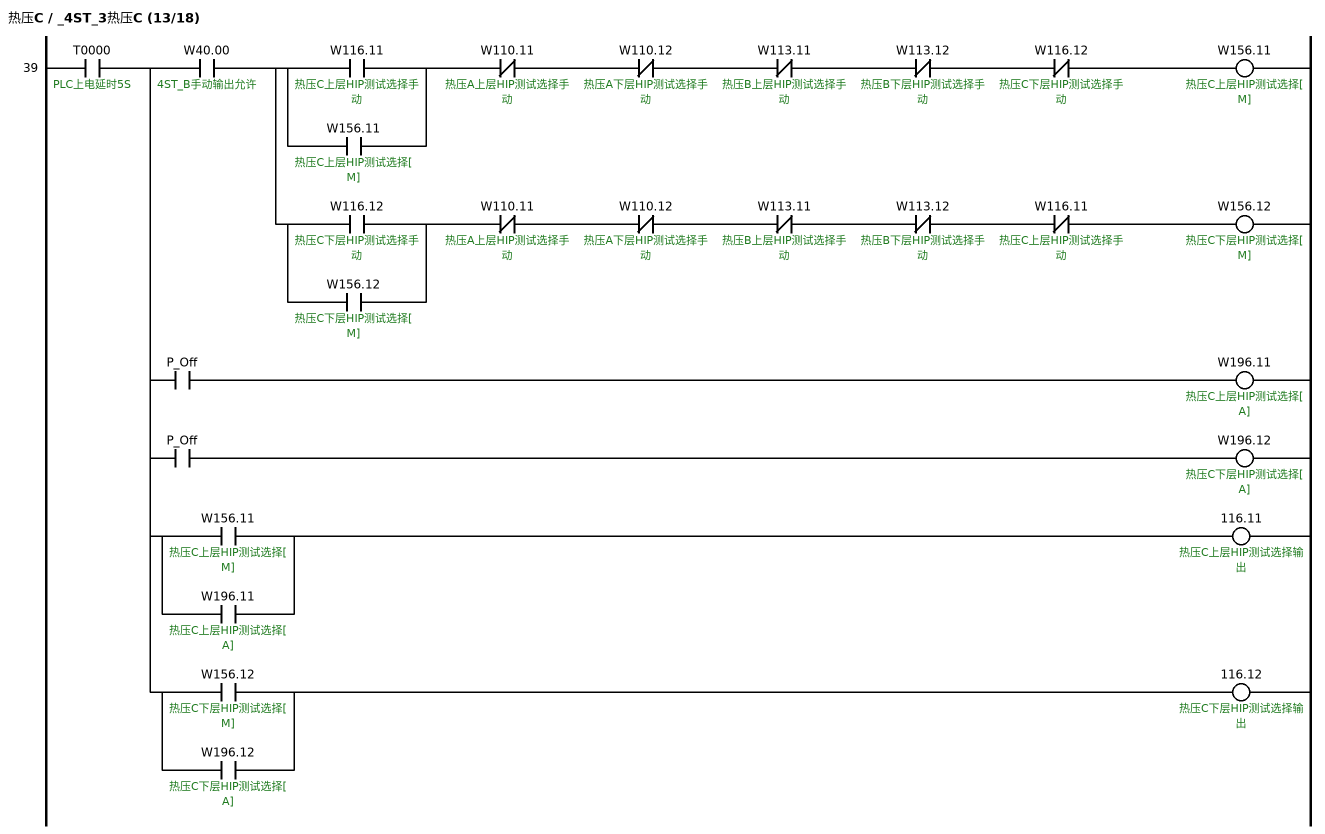
; rung 39
LD T0000  ; PLC上电延时5S
OUT TR0
AND W40.00  ; 4ST_B手动输出允许
OUT TR1
LD W116.11  ; 热压C上层HIP测试选择手动
OR W156.11  ; 热压C上层HIP测试选择[M]
ANDLD
ANDNOT W110.11  ; 热压A上层HIP测试选择手动
ANDNOT W110.12  ; 热压A下层HIP测试选择手动
ANDNOT W113.11  ; 热压B上层HIP测试选择手动
ANDNOT W113.12  ; 热压B下层HIP测试选择手动
ANDNOT W116.12  ; 热压C下层HIP测试选择手动
OUT W156.11  ; 热压C上层HIP测试选择[M]
LD TR1
LD W116.12  ; 热压C下层HIP测试选择手动
OR W156.12  ; 热压C下层HIP测试选择[M]
ANDLD
ANDNOT W110.11  ; 热压A上层HIP测试选择手动
ANDNOT W110.12  ; 热压A下层HIP测试选择手动
ANDNOT W113.11  ; 热压B上层HIP测试选择手动
ANDNOT W113.12  ; 热压B下层HIP测试选择手动
ANDNOT W116.11  ; 热压C上层HIP测试选择手动
OUT W156.12  ; 热压C下层HIP测试选择[M]
LD TR0
AND P_Off
OUT W196.11  ; 热压C上层HIP测试选择[A]
LD TR0
AND P_Off
OUT W196.12  ; 热压C下层HIP测试选择[A]
LD TR0
LD W156.11  ; 热压C上层HIP测试选择[M]
OR W196.11  ; 热压C上层HIP测试选择[A]
ANDLD
OUT 116.11  ; 热压C上层HIP测试选择输出
LD TR0
LD W156.12  ; 热压C下层HIP测试选择[M]
OR W196.12  ; 热压C下层HIP测试选择[A]
ANDLD
OUT 116.12  ; 热压C下层HIP测试选择输出

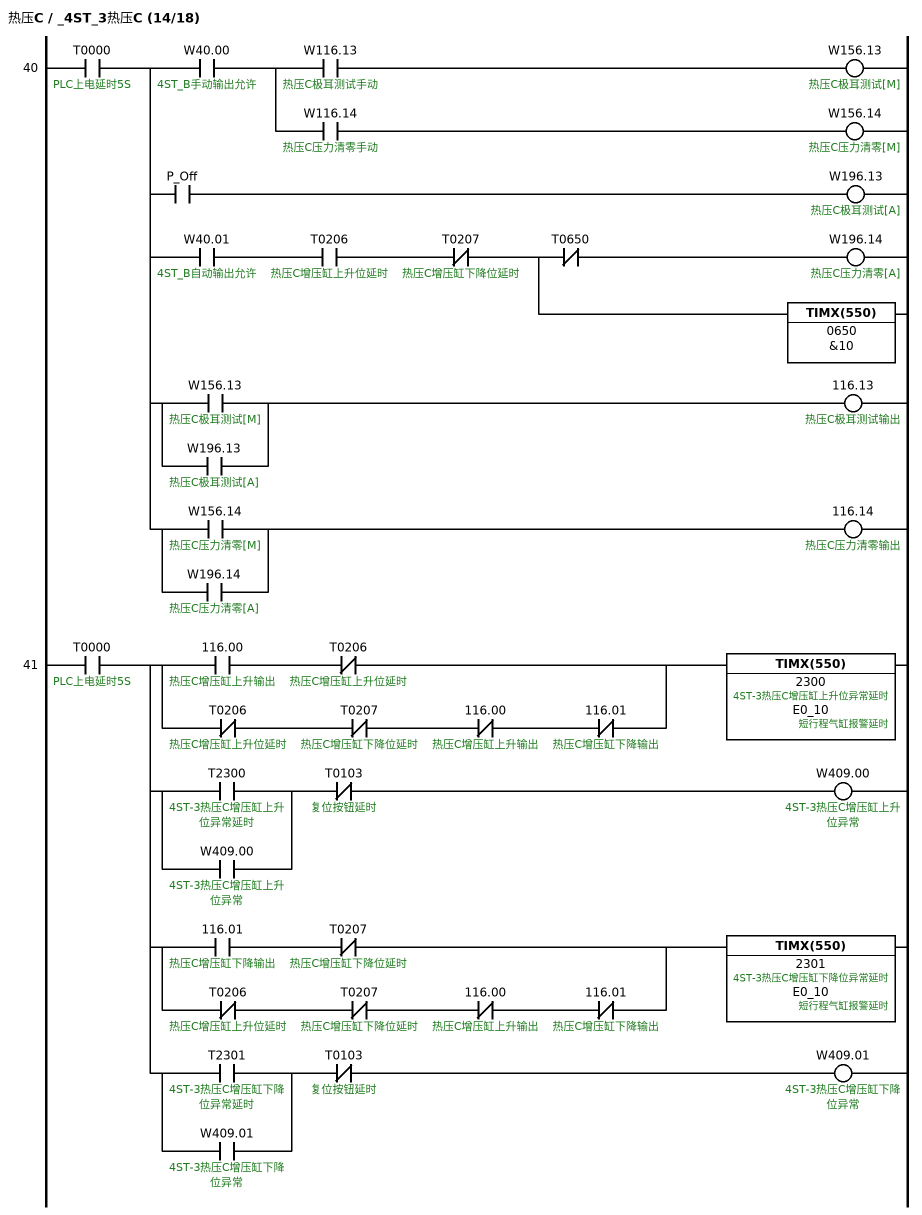
; rung 40
LD T0000  ; PLC上电延时5S
OUT TR0
AND W40.00  ; 4ST_B手动输出允许
OUT TR1
AND W116.13  ; 热压C极耳测试手动
OUT W156.13  ; 热压C极耳测试[M]
LD TR1
AND W116.14  ; 热压C压力清零手动
OUT W156.14  ; 热压C压力清零[M]
LD TR0
AND P_Off
OUT W196.13  ; 热压C极耳测试[A]
LD TR0
AND W40.01  ; 4ST_B自动输出允许
AND T0206  ; 热压C增压缸上升位延时
ANDNOT T0207  ; 热压C增压缸下降位延时
OUT TR1
ANDNOT T0650
OUT W196.14  ; 热压C压力清零[A]
LD TR1
TIMX(550) 0650 &10
LD TR0
LD W156.13  ; 热压C极耳测试[M]
OR W196.13  ; 热压C极耳测试[A]
ANDLD
OUT 116.13  ; 热压C极耳测试输出
LD TR0
LD W156.14  ; 热压C压力清零[M]
OR W196.14  ; 热压C压力清零[A]
ANDLD
OUT 116.14  ; 热压C压力清零输出
; rung 41
LD T0000  ; PLC上电延时5S
OUT TR0
LD 116.00  ; 热压C增压缸上升输出
ANDNOT T0206  ; 热压C增压缸上升位延时
LDNOT T0206  ; 热压C增压缸上升位延时
ANDNOT T0207  ; 热压C增压缸下降位延时
ANDNOT 116.00  ; 热压C增压缸上升输出
ANDNOT 116.01  ; 热压C增压缸下降输出
ORLD
ANDLD
TIMX(550) 2300 E0_10  ; 短行程气缸报警延时, 4ST-3热压C增压缸上升位异常延时
LD TR0
LD T2300  ; 4ST-3热压C增压缸上升位异常延时
OR W409.00  ; 4ST-3热压C增压缸上升位异常
ANDLD
ANDNOT T0103  ; 复位按钮延时
OUT W409.00  ; 4ST-3热压C增压缸上升位异常
LD TR0
LD 116.01  ; 热压C增压缸下降输出
ANDNOT T0207  ; 热压C增压缸下降位延时
LDNOT T0206  ; 热压C增压缸上升位延时
ANDNOT T0207  ; 热压C增压缸下降位延时
ANDNOT 116.00  ; 热压C增压缸上升输出
ANDNOT 116.01  ; 热压C增压缸下降输出
ORLD
ANDLD
TIMX(550) 2301 E0_10  ; 短行程气缸报警延时, 4ST-3热压C增压缸下降位异常延时
LD TR0
LD T2301  ; 4ST-3热压C增压缸下降位异常延时
OR W409.01  ; 4ST-3热压C增压缸下降位异常
ANDLD
ANDNOT T0103  ; 复位按钮延时
OUT W409.01  ; 4ST-3热压C增压缸下降位异常

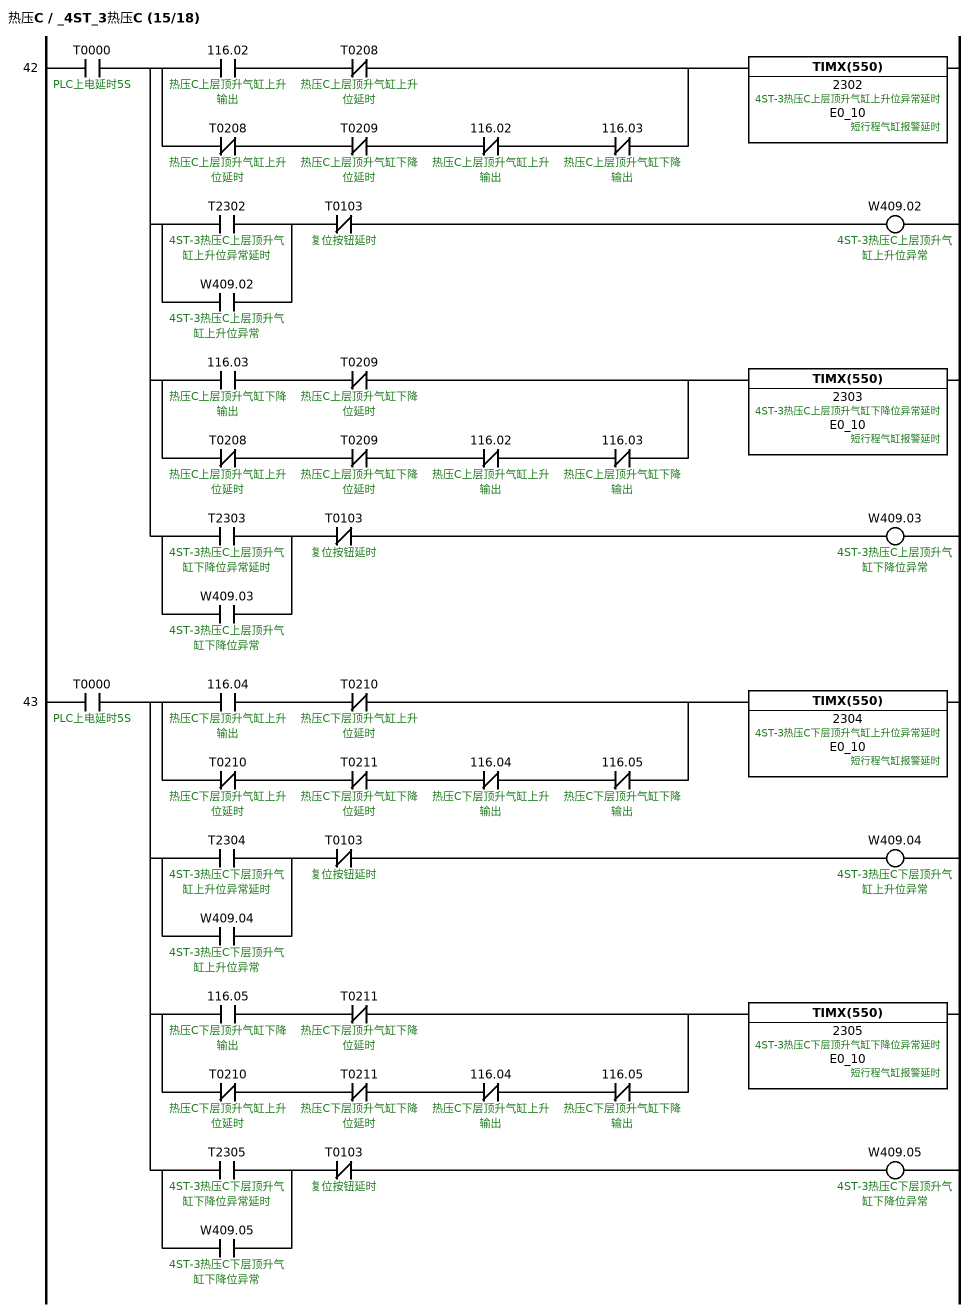
; rung 42
LD T0000  ; PLC上电延时5S
OUT TR0
LD 116.02  ; 热压C上层顶升气缸上升输出
ANDNOT T0208  ; 热压C上层顶升气缸上升位延时
LDNOT T0208  ; 热压C上层顶升气缸上升位延时
ANDNOT T0209  ; 热压C上层顶升气缸下降位延时
ANDNOT 116.02  ; 热压C上层顶升气缸上升输出
ANDNOT 116.03  ; 热压C上层顶升气缸下降输出
ORLD
ANDLD
TIMX(550) 2302 E0_10  ; 短行程气缸报警延时, 4ST-3热压C上层顶升气缸上升位异常延时
LD TR0
LD T2302  ; 4ST-3热压C上层顶升气缸上升位异常延时
OR W409.02  ; 4ST-3热压C上层顶升气缸上升位异常
ANDLD
ANDNOT T0103  ; 复位按钮延时
OUT W409.02  ; 4ST-3热压C上层顶升气缸上升位异常
LD TR0
LD 116.03  ; 热压C上层顶升气缸下降输出
ANDNOT T0209  ; 热压C上层顶升气缸下降位延时
LDNOT T0208  ; 热压C上层顶升气缸上升位延时
ANDNOT T0209  ; 热压C上层顶升气缸下降位延时
ANDNOT 116.02  ; 热压C上层顶升气缸上升输出
ANDNOT 116.03  ; 热压C上层顶升气缸下降输出
ORLD
ANDLD
TIMX(550) 2303 E0_10  ; 短行程气缸报警延时, 4ST-3热压C上层顶升气缸下降位异常延时
LD TR0
LD T2303  ; 4ST-3热压C上层顶升气缸下降位异常延时
OR W409.03  ; 4ST-3热压C上层顶升气缸下降位异常
ANDLD
ANDNOT T0103  ; 复位按钮延时
OUT W409.03  ; 4ST-3热压C上层顶升气缸下降位异常
; rung 43
LD T0000  ; PLC上电延时5S
OUT TR0
LD 116.04  ; 热压C下层顶升气缸上升输出
ANDNOT T0210  ; 热压C下层顶升气缸上升位延时
LDNOT T0210  ; 热压C下层顶升气缸上升位延时
ANDNOT T0211  ; 热压C下层顶升气缸下降位延时
ANDNOT 116.04  ; 热压C下层顶升气缸上升输出
ANDNOT 116.05  ; 热压C下层顶升气缸下降输出
ORLD
ANDLD
TIMX(550) 2304 E0_10  ; 短行程气缸报警延时, 4ST-3热压C下层顶升气缸上升位异常延时
LD TR0
LD T2304  ; 4ST-3热压C下层顶升气缸上升位异常延时
OR W409.04  ; 4ST-3热压C下层顶升气缸上升位异常
ANDLD
ANDNOT T0103  ; 复位按钮延时
OUT W409.04  ; 4ST-3热压C下层顶升气缸上升位异常
LD TR0
LD 116.05  ; 热压C下层顶升气缸下降输出
ANDNOT T0211  ; 热压C下层顶升气缸下降位延时
LDNOT T0210  ; 热压C下层顶升气缸上升位延时
ANDNOT T0211  ; 热压C下层顶升气缸下降位延时
ANDNOT 116.04  ; 热压C下层顶升气缸上升输出
ANDNOT 116.05  ; 热压C下层顶升气缸下降输出
ORLD
ANDLD
TIMX(550) 2305 E0_10  ; 短行程气缸报警延时, 4ST-3热压C下层顶升气缸下降位异常延时
LD TR0
LD T2305  ; 4ST-3热压C下层顶升气缸下降位异常延时
OR W409.05  ; 4ST-3热压C下层顶升气缸下降位异常
ANDLD
ANDNOT T0103  ; 复位按钮延时
OUT W409.05  ; 4ST-3热压C下层顶升气缸下降位异常

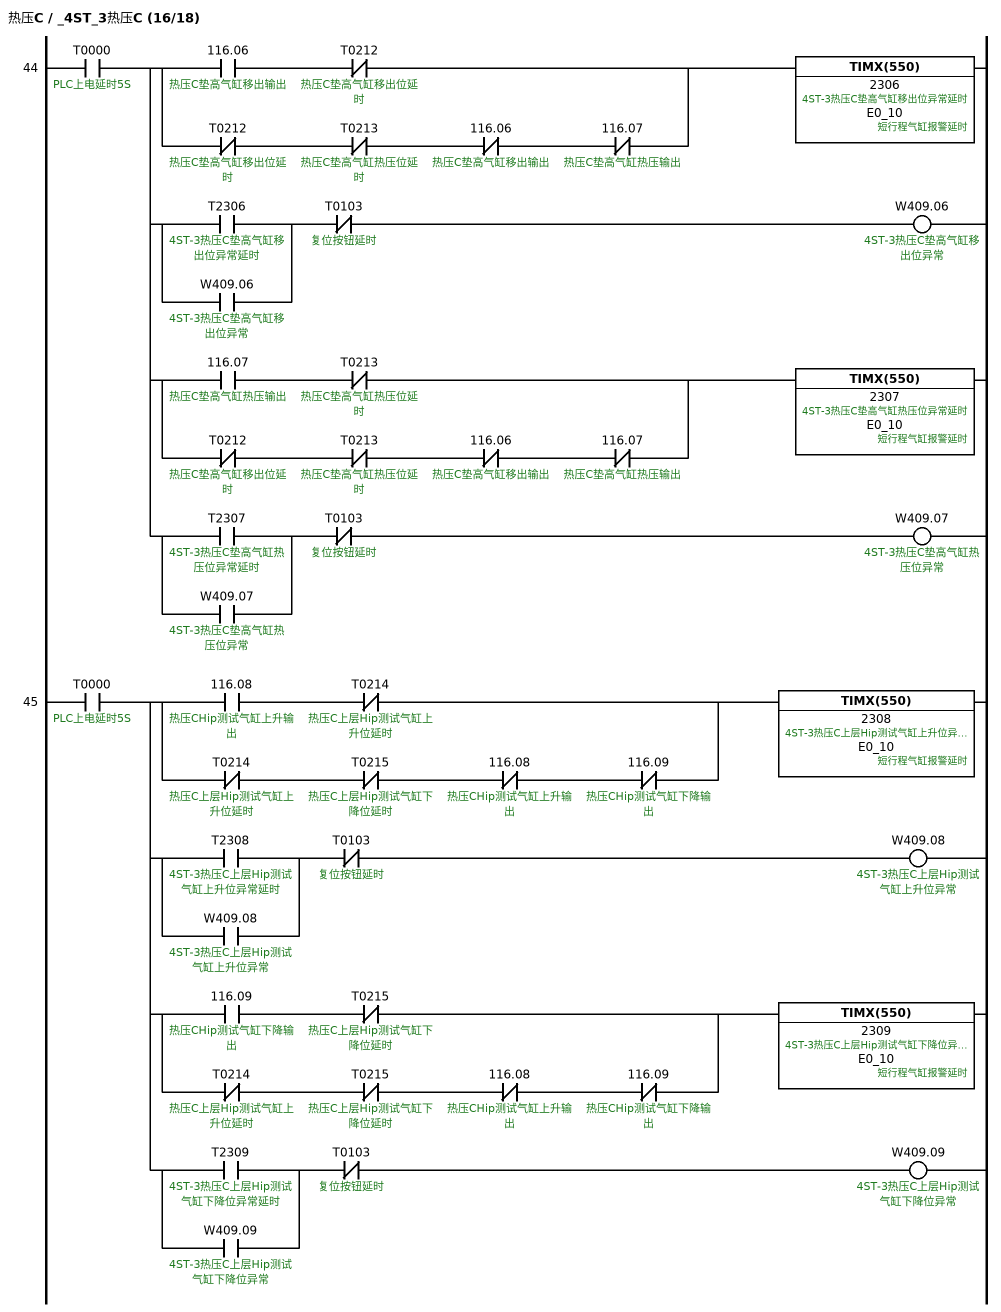
; rung 44
LD T0000  ; PLC上电延时5S
OUT TR0
LD 116.06  ; 热压C垫高气缸移出输出
ANDNOT T0212  ; 热压C垫高气缸移出位延时
LDNOT T0212  ; 热压C垫高气缸移出位延时
ANDNOT T0213  ; 热压C垫高气缸热压位延时
ANDNOT 116.06  ; 热压C垫高气缸移出输出
ANDNOT 116.07  ; 热压C垫高气缸热压输出
ORLD
ANDLD
TIMX(550) 2306 E0_10  ; 短行程气缸报警延时, 4ST-3热压C垫高气缸移出位异常延时
LD TR0
LD T2306  ; 4ST-3热压C垫高气缸移出位异常延时
OR W409.06  ; 4ST-3热压C垫高气缸移出位异常
ANDLD
ANDNOT T0103  ; 复位按钮延时
OUT W409.06  ; 4ST-3热压C垫高气缸移出位异常
LD TR0
LD 116.07  ; 热压C垫高气缸热压输出
ANDNOT T0213  ; 热压C垫高气缸热压位延时
LDNOT T0212  ; 热压C垫高气缸移出位延时
ANDNOT T0213  ; 热压C垫高气缸热压位延时
ANDNOT 116.06  ; 热压C垫高气缸移出输出
ANDNOT 116.07  ; 热压C垫高气缸热压输出
ORLD
ANDLD
TIMX(550) 2307 E0_10  ; 短行程气缸报警延时, 4ST-3热压C垫高气缸热压位异常延时
LD TR0
LD T2307  ; 4ST-3热压C垫高气缸热压位异常延时
OR W409.07  ; 4ST-3热压C垫高气缸热压位异常
ANDLD
ANDNOT T0103  ; 复位按钮延时
OUT W409.07  ; 4ST-3热压C垫高气缸热压位异常
; rung 45
LD T0000  ; PLC上电延时5S
OUT TR0
LD 116.08  ; 热压CHip测试气缸上升输出
ANDNOT T0214  ; 热压C上层Hip测试气缸上升位延时
LDNOT T0214  ; 热压C上层Hip测试气缸上升位延时
ANDNOT T0215  ; 热压C上层Hip测试气缸下降位延时
ANDNOT 116.08  ; 热压CHip测试气缸上升输出
ANDNOT 116.09  ; 热压CHip测试气缸下降输出
ORLD
ANDLD
TIMX(550) 2308 E0_10  ; 短行程气缸报警延时, 4ST-3热压C上层Hip测试气缸上升位异常延时
LD TR0
LD T2308  ; 4ST-3热压C上层Hip测试气缸上升位异常延时
OR W409.08  ; 4ST-3热压C上层Hip测试气缸上升位异常
ANDLD
ANDNOT T0103  ; 复位按钮延时
OUT W409.08  ; 4ST-3热压C上层Hip测试气缸上升位异常
LD TR0
LD 116.09  ; 热压CHip测试气缸下降输出
ANDNOT T0215  ; 热压C上层Hip测试气缸下降位延时
LDNOT T0214  ; 热压C上层Hip测试气缸上升位延时
ANDNOT T0215  ; 热压C上层Hip测试气缸下降位延时
ANDNOT 116.08  ; 热压CHip测试气缸上升输出
ANDNOT 116.09  ; 热压CHip测试气缸下降输出
ORLD
ANDLD
TIMX(550) 2309 E0_10  ; 短行程气缸报警延时, 4ST-3热压C上层Hip测试气缸下降位异常延时
LD TR0
LD T2309  ; 4ST-3热压C上层Hip测试气缸下降位异常延时
OR W409.09  ; 4ST-3热压C上层Hip测试气缸下降位异常
ANDLD
ANDNOT T0103  ; 复位按钮延时
OUT W409.09  ; 4ST-3热压C上层Hip测试气缸下降位异常

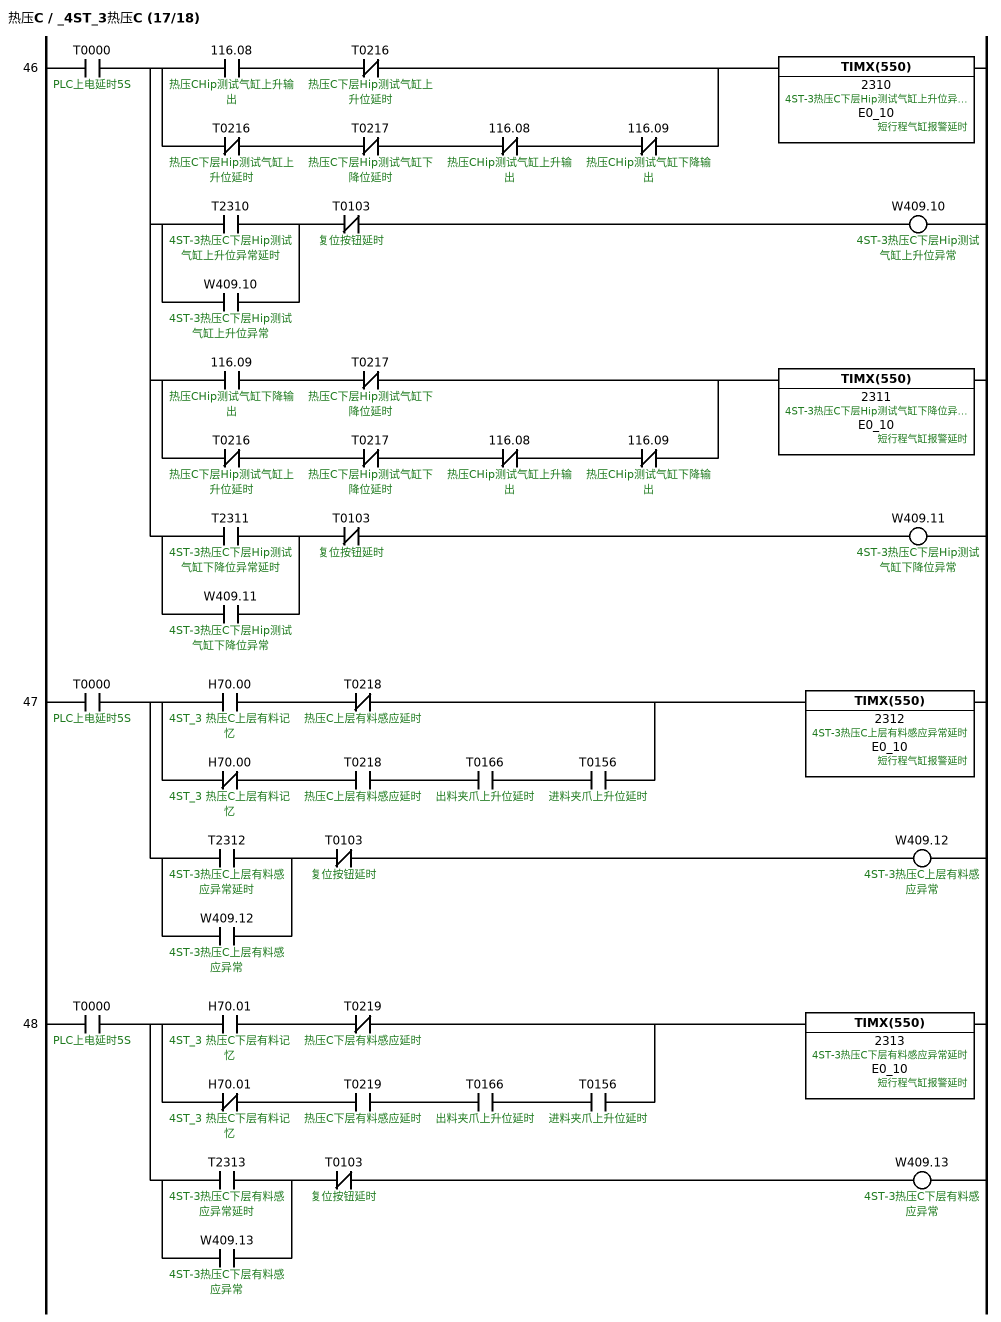
; rung 46
LD T0000  ; PLC上电延时5S
OUT TR0
LD 116.08  ; 热压CHip测试气缸上升输出
ANDNOT T0216  ; 热压C下层Hip测试气缸上升位延时
LDNOT T0216  ; 热压C下层Hip测试气缸上升位延时
ANDNOT T0217  ; 热压C下层Hip测试气缸下降位延时
ANDNOT 116.08  ; 热压CHip测试气缸上升输出
ANDNOT 116.09  ; 热压CHip测试气缸下降输出
ORLD
ANDLD
TIMX(550) 2310 E0_10  ; 短行程气缸报警延时, 4ST-3热压C下层Hip测试气缸上升位异常延时
LD TR0
LD T2310  ; 4ST-3热压C下层Hip测试气缸上升位异常延时
OR W409.10  ; 4ST-3热压C下层Hip测试气缸上升位异常
ANDLD
ANDNOT T0103  ; 复位按钮延时
OUT W409.10  ; 4ST-3热压C下层Hip测试气缸上升位异常
LD TR0
LD 116.09  ; 热压CHip测试气缸下降输出
ANDNOT T0217  ; 热压C下层Hip测试气缸下降位延时
LDNOT T0216  ; 热压C下层Hip测试气缸上升位延时
ANDNOT T0217  ; 热压C下层Hip测试气缸下降位延时
ANDNOT 116.08  ; 热压CHip测试气缸上升输出
ANDNOT 116.09  ; 热压CHip测试气缸下降输出
ORLD
ANDLD
TIMX(550) 2311 E0_10  ; 短行程气缸报警延时, 4ST-3热压C下层Hip测试气缸下降位异常延时
LD TR0
LD T2311  ; 4ST-3热压C下层Hip测试气缸下降位异常延时
OR W409.11  ; 4ST-3热压C下层Hip测试气缸下降位异常
ANDLD
ANDNOT T0103  ; 复位按钮延时
OUT W409.11  ; 4ST-3热压C下层Hip测试气缸下降位异常
; rung 47
LD T0000  ; PLC上电延时5S
OUT TR0
LD H70.00  ; 4ST_3 热压C上层有料记忆
ANDNOT T0218  ; 热压C上层有料感应延时
LDNOT H70.00  ; 4ST_3 热压C上层有料记忆
AND T0218  ; 热压C上层有料感应延时
AND T0166  ; 出料夹爪上升位延时
AND T0156  ; 进料夹爪上升位延时
ORLD
ANDLD
TIMX(550) 2312 E0_10  ; 短行程气缸报警延时, 4ST-3热压C上层有料感应异常延时
LD TR0
LD T2312  ; 4ST-3热压C上层有料感应异常延时
OR W409.12  ; 4ST-3热压C上层有料感应异常
ANDLD
ANDNOT T0103  ; 复位按钮延时
OUT W409.12  ; 4ST-3热压C上层有料感应异常
; rung 48
LD T0000  ; PLC上电延时5S
OUT TR0
LD H70.01  ; 4ST_3 热压C下层有料记忆
ANDNOT T0219  ; 热压C下层有料感应延时
LDNOT H70.01  ; 4ST_3 热压C下层有料记忆
AND T0219  ; 热压C下层有料感应延时
AND T0166  ; 出料夹爪上升位延时
AND T0156  ; 进料夹爪上升位延时
ORLD
ANDLD
TIMX(550) 2313 E0_10  ; 短行程气缸报警延时, 4ST-3热压C下层有料感应异常延时
LD TR0
LD T2313  ; 4ST-3热压C下层有料感应异常延时
OR W409.13  ; 4ST-3热压C下层有料感应异常
ANDLD
ANDNOT T0103  ; 复位按钮延时
OUT W409.13  ; 4ST-3热压C下层有料感应异常

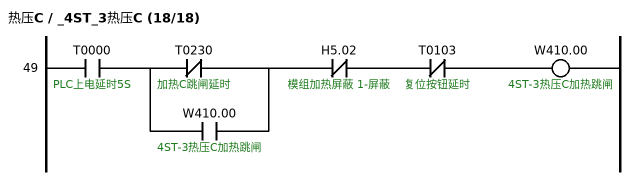
; rung 49
LD T0000  ; PLC上电延时5S
LDNOT T0230  ; 加热C跳闸延时
OR W410.00  ; 4ST-3热压C加热跳闸
ANDLD
ANDNOT H5.02  ; 模组加热屏蔽 1-屏蔽
ANDNOT T0103  ; 复位按钮延时
OUT W410.00  ; 4ST-3热压C加热跳闸

### Section 复位

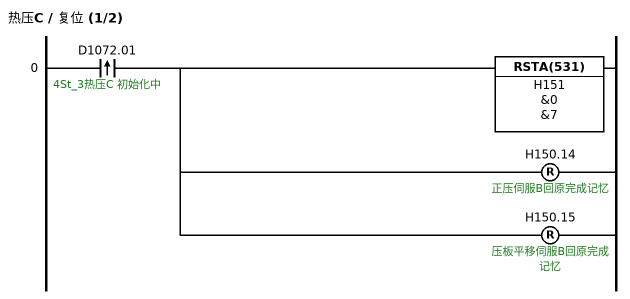
; rung 0
@LD D1072.01  ; 4St_3热压C 初始化中
RSTA(531) H151 &0 &7
RSET H150.14  ; 正压伺服B回原完成记忆
RSET H150.15  ; 压板平移伺服B回原完成记忆

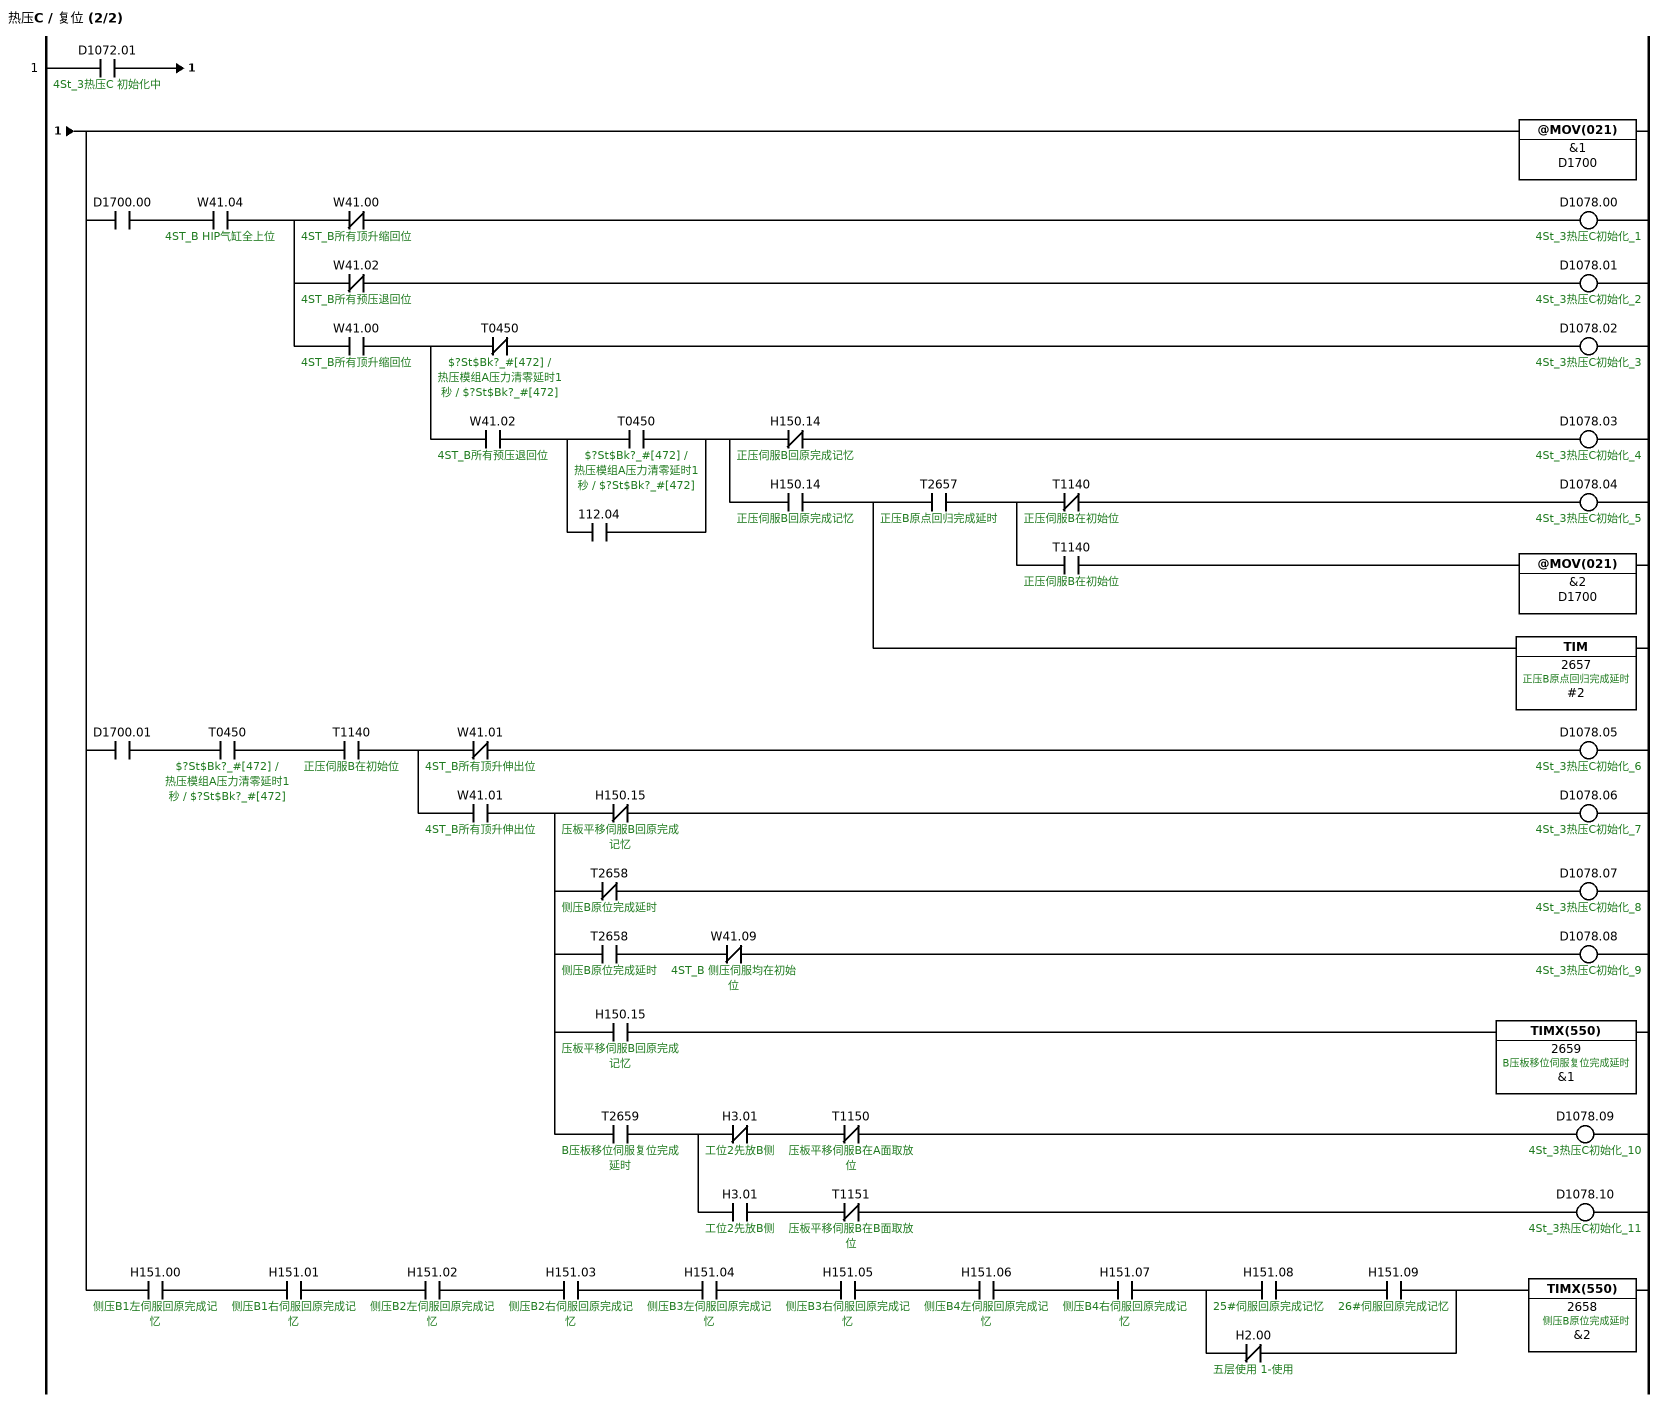
; rung 1
LD D1072.01  ; 4St_3热压C 初始化中
OUT TR0
@MOV(021) &1 D1700
AND D1700.00
AND W41.04  ; 4ST_B HIP气缸全上位
OUT TR1
ANDNOT W41.00  ; 4ST_B所有顶升缩回位
OUT D1078.00  ; 4St_3热压C初始化_1
LD TR1
ANDNOT W41.02  ; 4ST_B所有预压退回位
OUT D1078.01  ; 4St_3热压C初始化_2
LD TR1
AND W41.00  ; 4ST_B所有顶升缩回位
OUT TR1
ANDNOT T0450  ; $?St$Bk?_#[472] / 热压模组A压力清零延时1秒 / $?St$Bk?_#[472]
OUT D1078.02  ; 4St_3热压C初始化_3
LD TR1
AND W41.02  ; 4ST_B所有预压退回位
LD T0450  ; $?St$Bk?_#[472] / 热压模组A压力清零延时1秒 / $?St$Bk?_#[472]
OR 112.04
ANDLD
OUT TR1
ANDNOT H150.14  ; 正压伺服B回原完成记忆
OUT D1078.03  ; 4St_3热压C初始化_4
LD TR1
AND H150.14  ; 正压伺服B回原完成记忆
OUT TR1
AND T2657  ; 正压B原点回归完成延时
OUT TR2
ANDNOT T1140  ; 正压伺服B在初始位
OUT D1078.04  ; 4St_3热压C初始化_5
LD TR2
AND T1140  ; 正压伺服B在初始位
@MOV(021) &2 D1700
LD TR1
TIM 2657 #2  ; 正压B原点回归完成延时
LD TR0
AND D1700.01
AND T0450  ; $?St$Bk?_#[472] / 热压模组A压力清零延时1秒 / $?St$Bk?_#[472]
AND T1140  ; 正压伺服B在初始位
OUT TR1
ANDNOT W41.01  ; 4ST_B所有顶升伸出位
OUT D1078.05  ; 4St_3热压C初始化_6
LD TR1
AND W41.01  ; 4ST_B所有顶升伸出位
OUT TR1
ANDNOT H150.15  ; 压板平移伺服B回原完成记忆
OUT D1078.06  ; 4St_3热压C初始化_7
LD TR1
ANDNOT T2658  ; 侧压B原位完成延时
OUT D1078.07  ; 4St_3热压C初始化_8
LD TR1
AND T2658  ; 侧压B原位完成延时
ANDNOT W41.09  ; 4ST_B 侧压伺服均在初始位
OUT D1078.08  ; 4St_3热压C初始化_9
LD TR1
AND H150.15  ; 压板平移伺服B回原完成记忆
TIMX(550) 2659 &1  ; B压板移位伺服复位完成延时
LD TR1
AND T2659  ; B压板移位伺服复位完成延时
OUT TR1
ANDNOT H3.01  ; 工位2先放B侧
ANDNOT T1150  ; 压板平移伺服B在A面取放位
OUT D1078.09  ; 4St_3热压C初始化_10
LD TR1
AND H3.01  ; 工位2先放B侧
ANDNOT T1151  ; 压板平移伺服B在B面取放位
OUT D1078.10  ; 4St_3热压C初始化_11
LD TR0
AND H151.00  ; 侧压B1左伺服回原完成记忆
AND H151.01  ; 侧压B1右伺服回原完成记忆
AND H151.02  ; 侧压B2左伺服回原完成记忆
AND H151.03  ; 侧压B2右伺服回原完成记忆
AND H151.04  ; 侧压B3左伺服回原完成记忆
AND H151.05  ; 侧压B3右伺服回原完成记忆
AND H151.06  ; 侧压B4左伺服回原完成记忆
AND H151.07  ; 侧压B4右伺服回原完成记忆
LD H151.08  ; 25#伺服回原完成记忆
AND H151.09  ; 26#伺服回原完成记忆
ORNOT H2.00  ; 五层使用 1-使用
ANDLD
TIMX(550) 2658 &2  ; 侧压B原位完成延时

### Section 输出

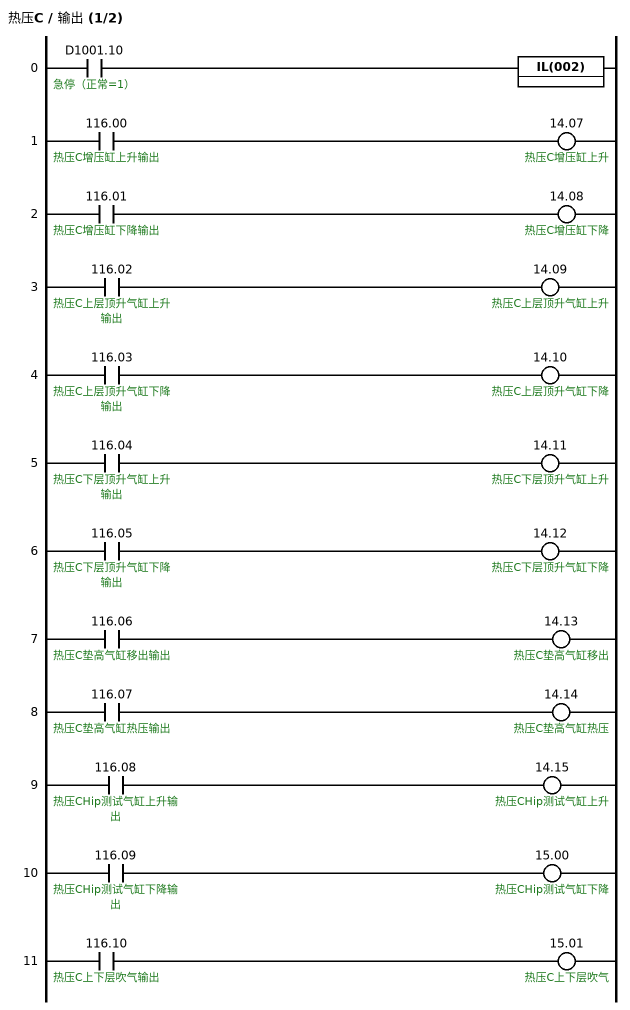
; rung 0
LD D1001.10  ; 急停（正常=1）
IL(002)
; rung 1
LD 116.00  ; 热压C增压缸上升输出
OUT 14.07  ; 热压C增压缸上升
; rung 2
LD 116.01  ; 热压C增压缸下降输出
OUT 14.08  ; 热压C增压缸下降
; rung 3
LD 116.02  ; 热压C上层顶升气缸上升输出
OUT 14.09  ; 热压C上层顶升气缸上升
; rung 4
LD 116.03  ; 热压C上层顶升气缸下降输出
OUT 14.10  ; 热压C上层顶升气缸下降
; rung 5
LD 116.04  ; 热压C下层顶升气缸上升输出
OUT 14.11  ; 热压C下层顶升气缸上升
; rung 6
LD 116.05  ; 热压C下层顶升气缸下降输出
OUT 14.12  ; 热压C下层顶升气缸下降
; rung 7
LD 116.06  ; 热压C垫高气缸移出输出
OUT 14.13  ; 热压C垫高气缸移出
; rung 8
LD 116.07  ; 热压C垫高气缸热压输出
OUT 14.14  ; 热压C垫高气缸热压
; rung 9
LD 116.08  ; 热压CHip测试气缸上升输出
OUT 14.15  ; 热压CHip测试气缸上升
; rung 10
LD 116.09  ; 热压CHip测试气缸下降输出
OUT 15.00  ; 热压CHip测试气缸下降
; rung 11
LD 116.10  ; 热压C上下层吹气输出
OUT 15.01  ; 热压C上下层吹气

